LIN {X 0,Y 446.444,Z 326.37,A -85,B 0,C 180,E1 -8665.154,E2 -8665.154} C_VEL
LIN {X 0,Y 446.485,Z 326.372,A -85,B 0,C 180,E1 -8668.179,E2 -8668.179} C_VEL
LIN {X 0,Y 446.42,Z 326.377,A -85,B 0,C 180,E1 -8671.775,E2 -8671.775} C_VEL
LIN {X 0,Y 446.43,Z 326.375,A -85,B 0,C 180,E1 -8674.523,E2 -8674.523} C_VEL
LIN {X 0,Y 446.417,Z 326.381,A -85,B 0,C 180,E1 -8678.08,E2 -8678.08} C_VEL
LIN {X 0,Y 446.439,Z 326.441,A -85,B 0,C 180,E1 -8680.92,E2 -8680.92} C_VEL
LIN {X 0,Y 446.853,Z 329.465,A -85,B 0,C 180,E1 -8683.791,E2 -8683.791} C_VEL
LIN {X 0,Y 447.265,Z 332.288,A -85,B 0,C 180,E1 -8686.288,E2 -8686.288} C_VEL
LIN {X 0,Y 447.313,Z 335.268,A -85,B 0,C 180,E1 -8688.709,E2 -8688.709} C_VEL
LIN {X 0,Y 447.118,Z 339.37,A -85,B 0,C 180,E1 -8691.807,E2 -8691.807} C_VEL
LIN {X 0,Y 446.836,Z 343.714,A -85,B 0,C 180,E1 -8694.873,E2 -8694.873} C_VEL
LIN {X 0,Y 446.563,Z 347.879,A -85,B 0,C 180,E1 -8697.65,E2 -8697.65} C_VEL
LIN {X 0,Y 446.282,Z 352.764,A -85,B 0,C 180,E1 -8700.779,E2 -8700.779} C_VEL
LIN {X 0,Y 446.038,Z 357.892,A -85,B 0,C 180,E1 -8703.913,E2 -8703.913} C_VEL
LIN {X 0,Y 445.811,Z 362.775,A -85,B 0,C 180,E1 -8706.789,E2 -8706.789} C_VEL
LIN {X 0,Y 445.645,Z 367.867,A -85,B 0,C 180,E1 -8709.699,E2 -8709.699} C_VEL
LIN {X 0,Y 445.513,Z 372.967,A -85,B 0,C 180,E1 -8712.559,E2 -8712.559} C_VEL
LIN {X 0,Y 445.479,Z 375.417,A -85,B 0,C 180,E1 -8713.876,E2 -8713.876} C_VEL
LIN {X 0,Y 447.43,Z 386.038,A -85,B 0,C 180,E1 -8714.246,E2 -8714.246} C_VEL
LIN {X 0,Y 448.77,Z 395.709,A -85,B 0,C 180,E1 -8714.676,E2 -8714.676} C_VEL
LIN {X 0,Y 449.202,Z 400.753,A -85,B 0,C 180,E1 -8714.924,E2 -8714.924} C_VEL
LIN {X 0,Y 448.604,Z 412.306,A -85,B 0,C 180,E1 -8715.599,E2 -8715.599} C_VEL
LIN {X 0,Y 448.106,Z 421.585,A -85,B 0,C 180,E1 -8716.278,E2 -8716.278} C_VEL
LIN {X 0,Y 447.61,Z 430.807,A -85,B 0,C 180,E1 -8717.099,E2 -8717.099} C_VEL
LIN {X 0,Y 447.187,Z 439.067,A -85,B 0,C 180,E1 -8717.981,E2 -8717.981} C_VEL
LIN {X 0,Y 446.718,Z 446.286,A -85,B 0,C 180,E1 -8718.888,E2 -8718.888} C_VEL
LIN {X 0,Y 446.391,Z 452.49,A -85,B 0,C 180,E1 -8719.798,E2 -8719.798} C_VEL
LIN {X 0,Y 446.032,Z 459.028,A -85,B 0,C 180,E1 -8720.934,E2 -8720.934} C_VEL
LIN {X 0,Y 445.849,Z 463.531,A -85,B 0,C 180,E1 -8721.844,E2 -8721.844} C_VEL
LIN {X 0,Y 445.576,Z 469.176,A -85,B 0,C 180,E1 -8723.252,E2 -8723.252} C_VEL
LIN {X 0,Y 445.485,Z 473.344,A -85,B 0,C 180,E1 -8724.568,E2 -8724.568} C_VEL
LIN {X 0,Y 445.415,Z 475.709,A -85,B 0,C 180,E1 -8725.475,E2 -8725.475} C_VEL
LIN {X 0,Y 445.433,Z 478.893,A -85,B 0,C 180,E1 -8727.287,E2 -8727.287} C_VEL
LIN {X 0,Y 445.356,Z 479.947,A -85,B 0,C 180,E1 -8728.191,E2 -8728.191} C_VEL
LIN {X 0,Y 445.339,Z 480.535,A -85,B 0,C 180,E1 -8729.096,E2 -8729.096} C_VEL
LIN {X 0,Y 445.339,Z 480.535,A -85,B 0,C 180,E1 -8730.904,E2 -8730.904} C_VEL
LIN {X 0,Y 445.356,Z 479.947,A -85,B 0,C 180,E1 -8731.809,E2 -8731.809} C_VEL
LIN {X 0,Y 445.433,Z 478.893,A -85,B 0,C 180,E1 -8732.713,E2 -8732.713} C_VEL
LIN {X 0,Y 445.415,Z 475.709,A -85,B 0,C 180,E1 -8734.525,E2 -8734.525} C_VEL
LIN {X 0,Y 445.488,Z 471.512,A -85,B 0,C 180,E1 -8736.065,E2 -8736.065} C_VEL
LIN {X 0,Y 445.668,Z 467.361,A -85,B 0,C 180,E1 -8737.248,E2 -8737.248} C_VEL
LIN {X 0,Y 445.96,Z 461.341,A -85,B 0,C 180,E1 -8738.61,E2 -8738.61} C_VEL
LIN {X 0,Y 446.221,Z 455.242,A -85,B 0,C 180,E1 -8739.748,E2 -8739.748} C_VEL
LIN {X 0,Y 446.523,Z 449.541,A -85,B 0,C 180,E1 -8740.657,E2 -8740.657} C_VEL
LIN {X 0,Y 447.057,Z 440.986,A -85,B 0,C 180,E1 -8741.792,E2 -8741.792} C_VEL
LIN {X 0,Y 447.521,Z 432.804,A -85,B 0,C 180,E1 -8742.701,E2 -8742.701} C_VEL
LIN {X 0,Y 447.897,Z 424.583,A -85,B 0,C 180,E1 -8743.472,E2 -8743.472} C_VEL
LIN {X 0,Y 448.394,Z 415.569,A -85,B 0,C 180,E1 -8744.176,E2 -8744.176} C_VEL
LIN {X 0,Y 448.9,Z 405.809,A -85,B 0,C 180,E1 -8744.797,E2 -8744.797} C_VEL
LIN {X 0,Y 449.135,Z 398.298,A -85,B 0,C 180,E1 -8745.195,E2 -8745.195} C_VEL
LIN {X 0,Y 447.528,Z 386.88,A -85,B 0,C 180,E1 -8745.722,E2 -8745.722} C_VEL
LIN {X 0,Y 445.555,Z 376.286,A -85,B 0,C 180,E1 -8746.101,E2 -8746.101} C_VEL
LIN {X 0,Y 445.479,Z 375.413,A -85,B 0,C 180,E1 -8746.126,E2 -8746.126} C_VEL
LIN {X 0,Y 445.613,Z 369.547,A -85,B 0,C 180,E1 -8749.342,E2 -8749.342} C_VEL
LIN {X 0,Y 445.748,Z 364.453,A -85,B 0,C 180,E1 -8752.235,E2 -8752.235} C_VEL
LIN {X 0,Y 445.93,Z 359.403,A -85,B 0,C 180,E1 -8755.184,E2 -8755.184} C_VEL
LIN {X 0,Y 446.214,Z 354.41,A -85,B 0,C 180,E1 -8758.197,E2 -8758.197} C_VEL
LIN {X 0,Y 446.473,Z 349.484,A -85,B 0,C 180,E1 -8761.296,E2 -8761.296} C_VEL
LIN {X 0,Y 446.764,Z 344.641,A -85,B 0,C 180,E1 -8764.493,E2 -8764.493} C_VEL
LIN {X 0,Y 447.042,Z 339.888,A -85,B 0,C 180,E1 -8767.815,E2 -8767.815} C_VEL
LIN {X 0,Y 447.292,Z 335.577,A -85,B 0,C 180,E1 -8771.045,E2 -8771.045} C_VEL
LIN {X 0,Y 447.366,Z 333.745,A -85,B 0,C 180,E1 -8772.494,E2 -8772.494} C_VEL
LIN {X 0,Y 447.054,Z 330.766,A -85,B 0,C 180,E1 -8775.026,E2 -8775.026} C_VEL
LIN {X 0,Y 446.512,Z 326.908,A -85,B 0,C 180,E1 -8778.618,E2 -8778.618} C_VEL
LIN {X 0,Y 446.439,Z 326.441,A -85,B 0,C 180,E1 -8779.08,E2 -8779.08} C_VEL
LIN {X 0,Y 446.417,Z 326.38,A -85,B 0,C 180,E1 -8781.92,E2 -8781.92} C_VEL
LIN {X 0,Y 446.43,Z 326.378,A -85,B 0,C 180,E1 -8785.477,E2 -8785.477} C_VEL
LIN {X 0,Y 446.416,Z 326.374,A -85,B 0,C 180,E1 -8788.699,E2 -8788.699} C_VEL
LIN {X 0,Y 446.485,Z 326.372,A -85,B 0,C 180,E1 -8791.821,E2 -8791.821} C_VEL
LIN {X 0,Y 446.444,Z 326.37,A -85,B 0,C 180,E1 -8794.846,E2 -8794.846} C_VEL
LIN {X 0,Y 446.448,Z 326.371,A -85,B 0,C 180,E1 -8798.245,E2 -8798.245} C_VEL
LIN {X 0,Y 446.453,Z 326.376,A -85,B 0,C 180,E1 -8801.649,E2 -8801.649} C_VEL
LIN {X 0,Y 446.509,Z 326.362,A -85,B 0,C 180,E1 -8804.479,E2 -8804.479} C_VEL
LIN {X 0,Y 446.518,Z 326.361,A -85,B 0,C 180,E1 -8808.193,E2 -8808.193} C_VEL
LIN {X 0,Y 446.6,Z 326.352,A -85,B 0,C 180,E1 -8811.857,E2 -8811.857} C_VEL
LIN {X 0,Y 446.642,Z 326.346,A -85,B 0,C 180,E1 -8814.582,E2 -8814.582} C_VEL
LIN {X 0,Y 446.707,Z 326.344,A -85,B 0,C 180,E1 -8817.294,E2 -8817.294} C_VEL
LIN {X 0,Y 446.792,Z 326.327,A -85,B 0,C 180,E1 -8820,E2 -8820} C_VEL
LIN {X 0,Y 446.708,Z 326.34,A -85,B 0,C 180,E1 -8822.705,E2 -8822.705} C_VEL
LIN {X 0,Y 446.638,Z 326.346,A -85,B 0,C 180,E1 -8826.323,E2 -8826.323} C_VEL
LIN {X 0,Y 446.536,Z 326.365,A -85,B 0,C 180,E1 -8829.055,E2 -8829.055} C_VEL
LIN {X 0,Y 446.52,Z 326.366,A -85,B 0,C 180,E1 -8832.729,E2 -8832.729} C_VEL
LIN {X 0,Y 446.494,Z 326.365,A -85,B 0,C 180,E1 -8836.227,E2 -8836.227} C_VEL
LIN {X 0,Y 446.467,Z 326.368,A -85,B 0,C 180,E1 -8839.303,E2 -8839.303} C_VEL
LIN {X 0,Y 446.416,Z 326.376,A -85,B 0,C 180,E1 -8842.199,E2 -8842.199} C_VEL
LIN {X 0,Y 446.454,Z 326.37,A -85,B 0,C 180,E1 -8845.152,E2 -8845.152} C_VEL
LIN {X 0,Y 446.482,Z 326.369,A -85,B 0,C 180,E1 -8848.178,E2 -8848.178} C_VEL
LIN {X 0,Y 446.417,Z 326.374,A -85,B 0,C 180,E1 -8851.775,E2 -8851.775} C_VEL
LIN {X 0,Y 446.427,Z 326.377,A -85,B 0,C 180,E1 -8854.522,E2 -8854.522} C_VEL
LIN {X 0,Y 446.432,Z 326.377,A -85,B 0,C 180,E1 -8858.082,E2 -8858.082} C_VEL
LIN {X 0,Y 446.444,Z 326.37,A -85,B 0,C 180,E1 -8860.92,E2 -8860.92} C_VEL
LIN {X 0,Y 446.442,Z 326.374,A -85,B 0,C 180,E1 -8863.84,E2 -8863.84} C_VEL
LIN {X 0,Y 446.395,Z 326.379,A -85,B 0,C 180,E1 -8866.403,E2 -8866.403} C_VEL
LIN {X 0,Y 446.464,Z 326.373,A -85,B 0,C 180,E1 -8869.805,E2 -8869.805} C_VEL
LIN {X 0,Y 446.428,Z 326.377,A -85,B 0,C 180,E1 -8872.123,E2 -8872.123} C_VEL
LIN {X 0,Y 446.427,Z 326.375,A -85,B 0,C 180,E1 -8875.477,E2 -8875.477} C_VEL
LIN {X 0,Y 446.413,Z 326.374,A -85,B 0,C 180,E1 -8878.7,E2 -8878.7} C_VEL
LIN {X 0,Y 446.481,Z 326.371,A -85,B 0,C 180,E1 -8881.821,E2 -8881.821} C_VEL
LIN {X 0,Y 446.454,Z 326.369,A -85,B 0,C 180,E1 -8884.848,E2 -8884.848} C_VEL
LIN {X 0,Y 446.444,Z 326.37,A -85,B 0,C 180,E1 -8888.245,E2 -8888.245} C_VEL
LIN {X 0,Y 446.454,Z 326.375,A -85,B 0,C 180,E1 -8891.649,E2 -8891.649} C_VEL
LIN {X 0,Y 446.505,Z 326.366,A -85,B 0,C 180,E1 -8894.48,E2 -8894.48} C_VEL
LIN {X 0,Y 446.514,Z 326.363,A -85,B 0,C 180,E1 -8898.193,E2 -8898.193} C_VEL
LIN {X 0,Y 446.597,Z 326.355,A -85,B 0,C 180,E1 -8901.858,E2 -8901.858} C_VEL
LIN {X 0,Y 446.644,Z 326.349,A -85,B 0,C 180,E1 -8904.583,E2 -8904.583} C_VEL
LIN {X 0,Y 446.616,Z 326.353,A -85,B 0,C 180,E1 -8906.99,E2 -8906.99} C_VEL
LIN {X 0,Y 446.098,Z 326.422,A -85,B 0,C 180,E1 -8907.742,E2 -8907.742} C_VEL
LIN {X 0,Y 443.285,Z 326.777,A -85,B 0,C 180,E1 -8908.965,E2 -8908.965} C_VEL
LIN {X 0,Y 440.802,Z 327.085,A -85,B 0,C 180,E1 -8909.952,E2 -8909.952} C_VEL
LIN {X 0,Y 439.714,Z 327.216,A -85,B 0,C 180,E1 -8910.716,E2 -8910.716} C_VEL
LIN {X 0,Y 439.619,Z 327.225,A -85,B 0,C 180,E1 -8910.975,E2 -8910.975} C_VEL
LIN {X 0,Y 439.653,Z 327.222,A -85,B 0,C 180,E1 -8912.749,E2 -8912.749} C_VEL
LIN {X 0,Y 439.616,Z 327.227,A -85,B 0,C 180,E1 -8916.425,E2 -8916.425} C_VEL
LIN {X 0,Y 439.497,Z 327.24,A -85,B 0,C 180,E1 -8919.202,E2 -8919.202} C_VEL
LIN {X 0,Y 439.462,Z 327.246,A -85,B 0,C 180,E1 -8922.938,E2 -8922.938} C_VEL
LIN {X 0,Y 439.444,Z 327.248,A -85,B 0,C 180,E1 -8926.349,E2 -8926.349} C_VEL
LIN {X 0,Y 439.399,Z 327.247,A -85,B 0,C 180,E1 -8929.626,E2 -8929.626} C_VEL
LIN {X 0,Y 439.361,Z 327.258,A -85,B 0,C 180,E1 -8932.576,E2 -8932.576} C_VEL
LIN {X 0,Y 439.401,Z 327.247,A -85,B 0,C 180,E1 -8935.585,E2 -8935.585} C_VEL
LIN {X 0,Y 439.414,Z 327.249,A -85,B 0,C 180,E1 -8938.674,E2 -8938.674} C_VEL
LIN {X 0,Y 439.367,Z 327.256,A -85,B 0,C 180,E1 -8942.031,E2 -8942.031} C_VEL
LIN {X 0,Y 439.392,Z 327.248,A -85,B 0,C 180,E1 -8945.341,E2 -8945.341} C_VEL
LIN {X 0,Y 439.392,Z 327.25,A -85,B 0,C 180,E1 -8948.594,E2 -8948.594} C_VEL
LIN {X 0,Y 439.395,Z 327.248,A -85,B 0,C 180,E1 -8951.259,E2 -8951.259} C_VEL
LIN {X 0,Y 439.401,Z 327.247,A -85,B 0,C 180,E1 -8954.729,E2 -8954.729} C_VEL
LIN {X 0,Y 439.409,Z 327.253,A -85,B 0,C 180,E1 -8957.798,E2 -8957.798} C_VEL
LIN {X 0,Y 439.446,Z 327.244,A -85,B 0,C 180,E1 -8960.23,E2 -8960.23} C_VEL
LIN {X 0,Y 439.372,Z 327.258,A -85,B 0,C 180,E1 -8963.713,E2 -8963.713} C_VEL
LIN {X 0,Y 439.369,Z 327.252,A -85,B 0,C 180,E1 -8967.054,E2 -8967.054} C_VEL
LIN {X 0,Y 439.379,Z 327.25,A -85,B 0,C 180,E1 -8970.275,E2 -8970.275} C_VEL
LIN {X 0,Y 439.426,Z 327.251,A -85,B 0,C 180,E1 -8973.397,E2 -8973.397} C_VEL
LIN {X 0,Y 439.383,Z 327.249,A -85,B 0,C 180,E1 -8976.43,E2 -8976.43} C_VEL
LIN {X 0,Y 439.387,Z 327.255,A -85,B 0,C 180,E1 -8979.398,E2 -8979.398} C_VEL
LIN {X 0,Y 439.429,Z 327.244,A -85,B 0,C 180,E1 -8982.31,E2 -8982.31} C_VEL
LIN {X 0,Y 439.446,Z 327.249,A -85,B 0,C 180,E1 -8985.174,E2 -8985.174} C_VEL
LIN {X 0,Y 439.482,Z 327.237,A -85,B 0,C 180,E1 -8988.002,E2 -8988.002} C_VEL
LIN {X 0,Y 439.547,Z 327.23,A -85,B 0,C 180,E1 -8991.727,E2 -8991.727} C_VEL
LIN {X 0,Y 439.616,Z 327.223,A -85,B 0,C 180,E1 -8994.496,E2 -8994.496} C_VEL
LIN {X 0,Y 439.635,Z 327.219,A -85,B 0,C 180,E1 -8998.168,E2 -8998.168} C_VEL
LIN {X 0,Y 439.761,Z 327.202,A -85,B 0,C 180,E1 -9000.001,E2 -9000.001} C_VEL
LIN {X 0,Y 439.654,Z 327.223,A -85,B 0,C 180,E1 -9002.749,E2 -9002.749} C_VEL
LIN {X 0,Y 439.611,Z 327.225,A -85,B 0,C 180,E1 -9006.426,E2 -9006.426} C_VEL
LIN {X 0,Y 439.5,Z 327.236,A -85,B 0,C 180,E1 -9009.202,E2 -9009.202} C_VEL
LIN {X 0,Y 439.466,Z 327.242,A -85,B 0,C 180,E1 -9012.938,E2 -9012.938} C_VEL
LIN {X 0,Y 439.446,Z 327.248,A -85,B 0,C 180,E1 -9016.349,E2 -9016.349} C_VEL
LIN {X 0,Y 439.402,Z 327.248,A -85,B 0,C 180,E1 -9019.627,E2 -9019.627} C_VEL
LIN {X 0,Y 439.364,Z 327.255,A -85,B 0,C 180,E1 -9022.576,E2 -9022.576} C_VEL
LIN {X 0,Y 439.398,Z 327.249,A -85,B 0,C 180,E1 -9025.586,E2 -9025.586} C_VEL
LIN {X 0,Y 439.418,Z 327.247,A -85,B 0,C 180,E1 -9028.674,E2 -9028.674} C_VEL
LIN {X 0,Y 439.371,Z 327.258,A -85,B 0,C 180,E1 -9032.031,E2 -9032.031} C_VEL
LIN {X 0,Y 439.395,Z 327.249,A -85,B 0,C 180,E1 -9035.341,E2 -9035.341} C_VEL
LIN {X 0,Y 439.384,Z 327.256,A -85,B 0,C 180,E1 -9038.595,E2 -9038.595} C_VEL
LIN {X 0,Y 439.407,Z 327.254,A -85,B 0,C 180,E1 -9039.85,E2 -9039.85} C_VEL
LIN {X 0,Y 439.501,Z 327.976,A -85,B 0,C 180,E1 -9041.274,E2 -9041.274} C_VEL
LIN {X 0,Y 439.994,Z 331.549,A -85,B 0,C 180,E1 -9044.653,E2 -9044.653} C_VEL
LIN {X 0,Y 440.322,Z 334.513,A -85,B 0,C 180,E1 -9047.241,E2 -9047.241} C_VEL
LIN {X 0,Y 440.206,Z 338.007,A -85,B 0,C 180,E1 -9050.026,E2 -9050.026} C_VEL
LIN {X 0,Y 439.988,Z 342.009,A -85,B 0,C 180,E1 -9053.003,E2 -9053.003} C_VEL
LIN {X 0,Y 439.663,Z 346.592,A -85,B 0,C 180,E1 -9056.225,E2 -9056.225} C_VEL
LIN {X 0,Y 439.366,Z 351.083,A -85,B 0,C 180,E1 -9059.212,E2 -9059.212} C_VEL
LIN {X 0,Y 439.085,Z 356.005,A -85,B 0,C 180,E1 -9062.343,E2 -9062.343} C_VEL
LIN {X 0,Y 438.83,Z 360.988,A -85,B 0,C 180,E1 -9065.393,E2 -9065.393} C_VEL
LIN {X 0,Y 438.634,Z 366.05,A -85,B 0,C 180,E1 -9068.376,E2 -9068.376} C_VEL
LIN {X 0,Y 438.492,Z 371.121,A -85,B 0,C 180,E1 -9071.304,E2 -9071.304} C_VEL
LIN {X 0,Y 438.405,Z 375.252,A -85,B 0,C 180,E1 -9073.607,E2 -9073.607} C_VEL
LIN {X 0,Y 440.56,Z 386.753,A -85,B 0,C 180,E1 -9074.025,E2 -9074.025} C_VEL
LIN {X 0,Y 442.111,Z 398.097,A -85,B 0,C 180,E1 -9074.558,E2 -9074.558} C_VEL
LIN {X 0,Y 442.181,Z 402.591,A -85,B 0,C 180,E1 -9074.796,E2 -9074.796} C_VEL
LIN {X 0,Y 441.714,Z 412.109,A -85,B 0,C 180,E1 -9075.37,E2 -9075.37} C_VEL
LIN {X 0,Y 441.183,Z 421.388,A -85,B 0,C 180,E1 -9076.058,E2 -9076.058} C_VEL
LIN {X 0,Y 440.702,Z 429.36,A -85,B 0,C 180,E1 -9076.764,E2 -9076.764} C_VEL
LIN {X 0,Y 440.364,Z 436.951,A -85,B 0,C 180,E1 -9077.558,E2 -9077.558} C_VEL
LIN {X 0,Y 439.732,Z 446.09,A -85,B 0,C 180,E1 -9078.709,E2 -9078.709} C_VEL
LIN {X 0,Y 439.369,Z 452.294,A -85,B 0,C 180,E1 -9079.633,E2 -9079.633} C_VEL
LIN {X 0,Y 438.994,Z 458.832,A -85,B 0,C 180,E1 -9080.788,E2 -9080.788} C_VEL
LIN {X 0,Y 438.783,Z 463.334,A -85,B 0,C 180,E1 -9081.712,E2 -9081.712} C_VEL
LIN {X 0,Y 438.515,Z 468.824,A -85,B 0,C 180,E1 -9083.096,E2 -9083.096} C_VEL
LIN {X 0,Y 438.385,Z 473.148,A -85,B 0,C 180,E1 -9084.48,E2 -9084.48} C_VEL
LIN {X 0,Y 438.344,Z 475.513,A -85,B 0,C 180,E1 -9085.402,E2 -9085.402} C_VEL
LIN {X 0,Y 438.341,Z 478.697,A -85,B 0,C 180,E1 -9087.243,E2 -9087.243} C_VEL
LIN {X 0,Y 438.279,Z 479.752,A -85,B 0,C 180,E1 -9088.162,E2 -9088.162} C_VEL
LIN {X 0,Y 438.252,Z 480.339,A -85,B 0,C 180,E1 -9089.081,E2 -9089.081} C_VEL
LIN {X 0,Y 438.252,Z 480.339,A -85,B 0,C 180,E1 -9090.919,E2 -9090.919} C_VEL
LIN {X 0,Y 438.279,Z 479.752,A -85,B 0,C 180,E1 -9091.838,E2 -9091.838} C_VEL
LIN {X 0,Y 438.341,Z 478.697,A -85,B 0,C 180,E1 -9092.757,E2 -9092.757} C_VEL
LIN {X 0,Y 438.345,Z 475.513,A -85,B 0,C 180,E1 -9094.598,E2 -9094.598} C_VEL
LIN {X 0,Y 438.445,Z 470.623,A -85,B 0,C 180,E1 -9096.37,E2 -9096.37} C_VEL
LIN {X 0,Y 438.681,Z 465.25,A -85,B 0,C 180,E1 -9097.827,E2 -9097.827} C_VEL
LIN {X 0,Y 438.944,Z 459.988,A -85,B 0,C 180,E1 -9098.981,E2 -9098.981} C_VEL
LIN {X 0,Y 439.282,Z 453.67,A -85,B 0,C 180,E1 -9100.136,E2 -9100.136} C_VEL
LIN {X 0,Y 439.609,Z 447.717,A -85,B 0,C 180,E1 -9101.06,E2 -9101.06} C_VEL
LIN {X 0,Y 440.086,Z 440.79,A -85,B 0,C 180,E1 -9101.982,E2 -9101.982} C_VEL
LIN {X 0,Y 440.579,Z 432.608,A -85,B 0,C 180,E1 -9102.904,E2 -9102.904} C_VEL
LIN {X 0,Y 441.031,Z 423.775,A -85,B 0,C 180,E1 -9103.739,E2 -9103.739} C_VEL
LIN {X 0,Y 441.518,Z 415.374,A -85,B 0,C 180,E1 -9104.401,E2 -9104.401} C_VEL
LIN {X 0,Y 442.038,Z 405.613,A -85,B 0,C 180,E1 -9105.032,E2 -9105.032} C_VEL
LIN {X 0,Y 442.279,Z 399.389,A -85,B 0,C 180,E1 -9105.377,E2 -9105.377} C_VEL
LIN {X 0,Y 440.596,Z 387.272,A -85,B 0,C 180,E1 -9105.956,E2 -9105.956} C_VEL
LIN {X 0,Y 438.525,Z 376.326,A -85,B 0,C 180,E1 -9106.36,E2 -9106.36} C_VEL
LIN {X 0,Y 438.404,Z 375.251,A -85,B 0,C 180,E1 -9106.394,E2 -9106.394} C_VEL
LIN {X 0,Y 438.539,Z 369.408,A -85,B 0,C 180,E1 -9109.666,E2 -9109.666} C_VEL
LIN {X 0,Y 438.694,Z 364.34,A -85,B 0,C 180,E1 -9112.612,E2 -9112.612} C_VEL
LIN {X 0,Y 438.903,Z 359.316,A -85,B 0,C 180,E1 -9115.616,E2 -9115.616} C_VEL
LIN {X 0,Y 439.164,Z 354.348,A -85,B 0,C 180,E1 -9118.691,E2 -9118.691} C_VEL
LIN {X 0,Y 439.483,Z 349.147,A -85,B 0,C 180,E1 -9122.053,E2 -9122.053} C_VEL
LIN {X 0,Y 439.782,Z 344.628,A -85,B 0,C 180,E1 -9125.121,E2 -9125.121} C_VEL
LIN {X 0,Y 440.086,Z 339.911,A -85,B 0,C 180,E1 -9128.522,E2 -9128.522} C_VEL
LIN {X 0,Y 440.336,Z 335.307,A -85,B 0,C 180,E1 -9132.093,E2 -9132.093} C_VEL
LIN {X 0,Y 440.083,Z 332.301,A -85,B 0,C 180,E1 -9134.641,E2 -9134.641} C_VEL
LIN {X 0,Y 439.638,Z 328.89,A -85,B 0,C 180,E1 -9137.824,E2 -9137.824} C_VEL
LIN {X 0,Y 439.462,Z 327.67,A -85,B 0,C 180,E1 -9139.028,E2 -9139.028} C_VEL
LIN {X 0,Y 439.431,Z 327.25,A -85,B 0,C 180,E1 -9140.227,E2 -9140.227} C_VEL
LIN {X 0,Y 439.374,Z 327.257,A -85,B 0,C 180,E1 -9143.712,E2 -9143.712} C_VEL
LIN {X 0,Y 439.373,Z 327.251,A -85,B 0,C 180,E1 -9147.054,E2 -9147.054} C_VEL
LIN {X 0,Y 439.383,Z 327.252,A -85,B 0,C 180,E1 -9150.274,E2 -9150.274} C_VEL
LIN {X 0,Y 439.428,Z 327.246,A -85,B 0,C 180,E1 -9153.396,E2 -9153.396} C_VEL
LIN {X 0,Y 439.384,Z 327.25,A -85,B 0,C 180,E1 -9156.429,E2 -9156.429} C_VEL
LIN {X 0,Y 439.388,Z 327.253,A -85,B 0,C 180,E1 -9159.397,E2 -9159.397} C_VEL
LIN {X 0,Y 439.406,Z 327.247,A -85,B 0,C 180,E1 -9162.308,E2 -9162.308} C_VEL
LIN {X 0,Y 439.449,Z 327.244,A -85,B 0,C 180,E1 -9165.174,E2 -9165.174} C_VEL
LIN {X 0,Y 439.484,Z 327.238,A -85,B 0,C 180,E1 -9168.001,E2 -9168.001} C_VEL
LIN {X 0,Y 439.548,Z 327.232,A -85,B 0,C 180,E1 -9171.726,E2 -9171.726} C_VEL
LIN {X 0,Y 439.617,Z 327.22,A -85,B 0,C 180,E1 -9174.495,E2 -9174.495} C_VEL
LIN {X 0,Y 439.634,Z 327.218,A -85,B 0,C 180,E1 -9178.167,E2 -9178.167} C_VEL
LIN {X 0,Y 439.761,Z 327.202,A -85,B 0,C 180,E1 -9179.999,E2 -9179.999} C_VEL
LIN {X 0,Y 439.655,Z 327.219,A -85,B 0,C 180,E1 -9182.748,E2 -9182.748} C_VEL
LIN {X 0,Y 439.598,Z 327.223,A -85,B 0,C 180,E1 -9186.566,E2 -9186.566} C_VEL
LIN {X 0,Y 439.498,Z 327.239,A -85,B 0,C 180,E1 -9189.201,E2 -9189.201} C_VEL
LIN {X 0,Y 439.464,Z 327.246,A -85,B 0,C 180,E1 -9192.937,E2 -9192.937} C_VEL
LIN {X 0,Y 439.445,Z 327.244,A -85,B 0,C 180,E1 -9196.348,E2 -9196.348} C_VEL
LIN {X 0,Y 439.4,Z 327.247,A -85,B 0,C 180,E1 -9199.626,E2 -9199.626} C_VEL
LIN {X 0,Y 439.362,Z 327.259,A -85,B 0,C 180,E1 -9202.575,E2 -9202.575} C_VEL
LIN {X 0,Y 439.402,Z 327.247,A -85,B 0,C 180,E1 -9205.584,E2 -9205.584} C_VEL
LIN {X 0,Y 439.414,Z 327.251,A -85,B 0,C 180,E1 -9208.673,E2 -9208.673} C_VEL
LIN {X 0,Y 439.368,Z 327.254,A -85,B 0,C 180,E1 -9212.03,E2 -9212.03} C_VEL
LIN {X 0,Y 439.393,Z 327.248,A -85,B 0,C 180,E1 -9215.34,E2 -9215.34} C_VEL
LIN {X 0,Y 439.392,Z 327.251,A -85,B 0,C 180,E1 -9218.593,E2 -9218.593} C_VEL
LIN {X 0,Y 439.401,Z 327.247,A -85,B 0,C 180,E1 -9221.259,E2 -9221.259} C_VEL
LIN {X 0,Y 439.405,Z 327.248,A -85,B 0,C 180,E1 -9224.728,E2 -9224.728} C_VEL
LIN {X 0,Y 439.394,Z 327.253,A -85,B 0,C 180,E1 -9227.796,E2 -9227.796} C_VEL
LIN {X 0,Y 439.445,Z 327.246,A -85,B 0,C 180,E1 -9230.23,E2 -9230.23} C_VEL
LIN {X 0,Y 439.373,Z 327.256,A -85,B 0,C 180,E1 -9233.713,E2 -9233.713} C_VEL
LIN {X 0,Y 439.368,Z 327.252,A -85,B 0,C 180,E1 -9237.054,E2 -9237.054} C_VEL
LIN {X 0,Y 439.379,Z 327.251,A -85,B 0,C 180,E1 -9240.274,E2 -9240.274} C_VEL
LIN {X 0,Y 439.426,Z 327.248,A -85,B 0,C 180,E1 -9243.396,E2 -9243.396} C_VEL
LIN {X 0,Y 439.382,Z 327.249,A -85,B 0,C 180,E1 -9246.429,E2 -9246.429} C_VEL
LIN {X 0,Y 439.386,Z 327.255,A -85,B 0,C 180,E1 -9249.397,E2 -9249.397} C_VEL
LIN {X 0,Y 439.428,Z 327.247,A -85,B 0,C 180,E1 -9252.309,E2 -9252.309} C_VEL
LIN {X 0,Y 439.446,Z 327.248,A -85,B 0,C 180,E1 -9255.174,E2 -9255.174} C_VEL
LIN {X 0,Y 439.48,Z 327.24,A -85,B 0,C 180,E1 -9258.001,E2 -9258.001} C_VEL
LIN {X 0,Y 439.545,Z 327.234,A -85,B 0,C 180,E1 -9261.726,E2 -9261.726} C_VEL
LIN {X 0,Y 439.619,Z 327.224,A -85,B 0,C 180,E1 -9264.496,E2 -9264.496} C_VEL
LIN {X 0,Y 439.633,Z 327.222,A -85,B 0,C 180,E1 -9268.168,E2 -9268.168} C_VEL
LIN {X 0,Y 439.761,Z 327.207,A -85,B 0,C 180,E1 -9270,E2 -9270} C_VEL
LIN {X 0,Y 439.619,Z 327.225,A -85,B 0,C 180,E1 -9270.975,E2 -9270.975} C_VEL
LIN {X 0,Y 438.902,Z 327.313,A -85,B 0,C 180,E1 -9271.739,E2 -9271.739} C_VEL
LIN {X 0,Y 435.923,Z 327.686,A -85,B 0,C 180,E1 -9272.978,E2 -9272.978} C_VEL
LIN {X 0,Y 433.471,Z 327.992,A -85,B 0,C 180,E1 -9273.978,E2 -9273.978} C_VEL
LIN {X 0,Y 432.497,Z 328.113,A -85,B 0,C 180,E1 -9274.753,E2 -9274.753} C_VEL
LIN {X 0,Y 432.46,Z 328.115,A -85,B 0,C 180,E1 -9275.015,E2 -9275.015} C_VEL
LIN {X 0,Y 432.582,Z 328.101,A -85,B 0,C 180,E1 -9277.679,E2 -9277.679} C_VEL
LIN {X 0,Y 432.39,Z 328.125,A -85,B 0,C 180,E1 -9281.247,E2 -9281.247} C_VEL
LIN {X 0,Y 432.371,Z 328.128,A -85,B 0,C 180,E1 -9284.112,E2 -9284.112} C_VEL
LIN {X 0,Y 432.394,Z 328.126,A -85,B 0,C 180,E1 -9287.012,E2 -9287.012} C_VEL
LIN {X 0,Y 432.335,Z 328.129,A -85,B 0,C 180,E1 -9289.96,E2 -9289.96} C_VEL
LIN {X 0,Y 432.315,Z 328.132,A -85,B 0,C 180,E1 -9292.964,E2 -9292.964} C_VEL
LIN {X 0,Y 432.361,Z 328.128,A -85,B 0,C 180,E1 -9296.033,E2 -9296.033} C_VEL
LIN {X 0,Y 432.339,Z 328.127,A -85,B 0,C 180,E1 -9299.188,E2 -9299.188} C_VEL
LIN {X 0,Y 432.319,Z 328.134,A -85,B 0,C 180,E1 -9302.443,E2 -9302.443} C_VEL
LIN {X 0,Y 432.342,Z 328.128,A -85,B 0,C 180,E1 -9305.632,E2 -9305.632} C_VEL
LIN {X 0,Y 432.354,Z 328.126,A -85,B 0,C 180,E1 -9308.718,E2 -9308.718} C_VEL
LIN {X 0,Y 432.362,Z 328.129,A -85,B 0,C 180,E1 -9311.793,E2 -9311.793} C_VEL
LIN {X 0,Y 432.375,Z 328.127,A -85,B 0,C 180,E1 -9315.659,E2 -9315.659} C_VEL
LIN {X 0,Y 432.37,Z 328.124,A -85,B 0,C 180,E1 -9318.392,E2 -9318.392} C_VEL
LIN {X 0,Y 432.347,Z 328.132,A -85,B 0,C 180,E1 -9321.852,E2 -9321.852} C_VEL
LIN {X 0,Y 432.336,Z 328.131,A -85,B 0,C 180,E1 -9325.323,E2 -9325.323} C_VEL
LIN {X 0,Y 432.319,Z 328.129,A -85,B 0,C 180,E1 -9328.654,E2 -9328.654} C_VEL
LIN {X 0,Y 432.379,Z 328.125,A -85,B 0,C 180,E1 -9331.877,E2 -9331.877} C_VEL
LIN {X 0,Y 432.349,Z 328.128,A -85,B 0,C 180,E1 -9334.999,E2 -9334.999} C_VEL
LIN {X 0,Y 432.355,Z 328.125,A -85,B 0,C 180,E1 -9338.046,E2 -9338.046} C_VEL
LIN {X 0,Y 432.384,Z 328.125,A -85,B 0,C 180,E1 -9341.03,E2 -9341.03} C_VEL
LIN {X 0,Y 432.429,Z 328.116,A -85,B 0,C 180,E1 -9343.962,E2 -9343.962} C_VEL
LIN {X 0,Y 432.457,Z 328.113,A -85,B 0,C 180,E1 -9347.804,E2 -9347.804} C_VEL
LIN {X 0,Y 432.491,Z 328.109,A -85,B 0,C 180,E1 -9351.591,E2 -9351.591} C_VEL
LIN {X 0,Y 432.593,Z 328.097,A -85,B 0,C 180,E1 -9354.407,E2 -9354.407} C_VEL
LIN {X 0,Y 432.605,Z 328.094,A -85,B 0,C 180,E1 -9358.139,E2 -9358.139} C_VEL
LIN {X 0,Y 432.731,Z 328.078,A -85,B 0,C 180,E1 -9360.001,E2 -9360.001} C_VEL
LIN {X 0,Y 432.603,Z 328.101,A -85,B 0,C 180,E1 -9362.794,E2 -9362.794} C_VEL
LIN {X 0,Y 432.564,Z 328.105,A -85,B 0,C 180,E1 -9366.531,E2 -9366.531} C_VEL
LIN {X 0,Y 432.443,Z 328.114,A -85,B 0,C 180,E1 -9369.354,E2 -9369.354} C_VEL
LIN {X 0,Y 432.431,Z 328.119,A -85,B 0,C 180,E1 -9372.804,E2 -9372.804} C_VEL
LIN {X 0,Y 432.412,Z 328.125,A -85,B 0,C 180,E1 -9376.479,E2 -9376.479} C_VEL
LIN {X 0,Y 432.338,Z 328.13,A -85,B 0,C 180,E1 -9379.961,E2 -9379.961} C_VEL
LIN {X 0,Y 432.318,Z 328.13,A -85,B 0,C 180,E1 -9382.965,E2 -9382.965} C_VEL
LIN {X 0,Y 432.361,Z 328.13,A -85,B 0,C 180,E1 -9386.033,E2 -9386.033} C_VEL
LIN {X 0,Y 432.343,Z 328.126,A -85,B 0,C 180,E1 -9389.188,E2 -9389.188} C_VEL
LIN {X 0,Y 432.324,Z 328.131,A -85,B 0,C 180,E1 -9392.443,E2 -9392.443} C_VEL
LIN {X 0,Y 432.345,Z 328.13,A -85,B 0,C 180,E1 -9395.632,E2 -9395.632} C_VEL
LIN {X 0,Y 432.351,Z 328.132,A -85,B 0,C 180,E1 -9399.343,E2 -9399.343} C_VEL
LIN {X 0,Y 432.351,Z 328.132,A -85,B 0,C 180,E1 -9400.182,E2 -9400.182} C_VEL
LIN {X 0,Y 432.739,Z 330.94,A -85,B 0,C 180,E1 -9403.044,E2 -9403.044} C_VEL
LIN {X 0,Y 433.184,Z 333.88,A -85,B 0,C 180,E1 -9405.763,E2 -9405.763} C_VEL
LIN {X 0,Y 433.293,Z 336.882,A -85,B 0,C 180,E1 -9408.317,E2 -9408.317} C_VEL
LIN {X 0,Y 433.082,Z 340.511,A -85,B 0,C 180,E1 -9411.164,E2 -9411.164} C_VEL
LIN {X 0,Y 432.821,Z 344.703,A -85,B 0,C 180,E1 -9414.281,E2 -9414.281} C_VEL
LIN {X 0,Y 432.463,Z 349.581,A -85,B 0,C 180,E1 -9417.679,E2 -9417.679} C_VEL
LIN {X 0,Y 432.154,Z 354.289,A -85,B 0,C 180,E1 -9420.799,E2 -9420.799} C_VEL
LIN {X 0,Y 431.901,Z 359.229,A -85,B 0,C 180,E1 -9423.938,E2 -9423.938} C_VEL
LIN {X 0,Y 431.649,Z 364.228,A -85,B 0,C 180,E1 -9426.998,E2 -9426.998} C_VEL
LIN {X 0,Y 431.461,Z 369.271,A -85,B 0,C 180,E1 -9429.997,E2 -9429.997} C_VEL
LIN {X 0,Y 431.336,Z 375.07,A -85,B 0,C 180,E1 -9433.329,E2 -9433.329} C_VEL
LIN {X 0,Y 433.398,Z 386.39,A -85,B 0,C 180,E1 -9433.748,E2 -9433.748} C_VEL
LIN {X 0,Y 434.885,Z 396.601,A -85,B 0,C 180,E1 -9434.235,E2 -9434.235} C_VEL
LIN {X 0,Y 435.434,Z 401.389,A -85,B 0,C 180,E1 -9434.495,E2 -9434.495} C_VEL
LIN {X 0,Y 434.828,Z 411.913,A -85,B 0,C 180,E1 -9435.133,E2 -9435.133} C_VEL
LIN {X 0,Y 434.286,Z 421.192,A -85,B 0,C 180,E1 -9435.832,E2 -9435.832} C_VEL
LIN {X 0,Y 433.717,Z 429.983,A -85,B 0,C 180,E1 -9436.633,E2 -9436.633} C_VEL
LIN {X 0,Y 433.279,Z 438.674,A -85,B 0,C 180,E1 -9437.589,E2 -9437.589} C_VEL
LIN {X 0,Y 432.758,Z 445.894,A -85,B 0,C 180,E1 -9438.525,E2 -9438.525} C_VEL
LIN {X 0,Y 432.348,Z 452.097,A -85,B 0,C 180,E1 -9439.463,E2 -9439.463} C_VEL
LIN {X 0,Y 431.952,Z 458.635,A -85,B 0,C 180,E1 -9440.636,E2 -9440.636} C_VEL
LIN {X 0,Y 431.721,Z 463.137,A -85,B 0,C 180,E1 -9441.575,E2 -9441.575} C_VEL
LIN {X 0,Y 431.437,Z 468.628,A -85,B 0,C 180,E1 -9442.982,E2 -9442.982} C_VEL
LIN {X 0,Y 431.288,Z 472.951,A -85,B 0,C 180,E1 -9444.389,E2 -9444.389} C_VEL
LIN {X 0,Y 431.274,Z 475.318,A -85,B 0,C 180,E1 -9445.326,E2 -9445.326} C_VEL
LIN {X 0,Y 431.236,Z 478.501,A -85,B 0,C 180,E1 -9447.198,E2 -9447.198} C_VEL
LIN {X 0,Y 431.203,Z 479.557,A -85,B 0,C 180,E1 -9448.132,E2 -9448.132} C_VEL
LIN {X 0,Y 431.169,Z 480.144,A -85,B 0,C 180,E1 -9449.066,E2 -9449.066} C_VEL
LIN {X 0,Y 431.169,Z 480.144,A -85,B 0,C 180,E1 -9450.934,E2 -9450.934} C_VEL
LIN {X 0,Y 431.203,Z 479.557,A -85,B 0,C 180,E1 -9451.868,E2 -9451.868} C_VEL
LIN {X 0,Y 431.188,Z 477.113,A -85,B 0,C 180,E1 -9453.738,E2 -9453.738} C_VEL
LIN {X 0,Y 431.299,Z 474.168,A -85,B 0,C 180,E1 -9455.142,E2 -9455.142} C_VEL
LIN {X 0,Y 431.378,Z 470.181,A -85,B 0,C 180,E1 -9456.548,E2 -9456.548} C_VEL
LIN {X 0,Y 431.608,Z 465.053,A -85,B 0,C 180,E1 -9457.956,E2 -9457.956} C_VEL
LIN {X 0,Y 431.881,Z 459.79,A -85,B 0,C 180,E1 -9459.129,E2 -9459.129} C_VEL
LIN {X 0,Y 432.248,Z 453.473,A -85,B 0,C 180,E1 -9460.303,E2 -9460.303} C_VEL
LIN {X 0,Y 432.626,Z 447.52,A -85,B 0,C 180,E1 -9461.241,E2 -9461.241} C_VEL
LIN {X 0,Y 433.13,Z 440.594,A -85,B 0,C 180,E1 -9462.177,E2 -9462.177} C_VEL
LIN {X 0,Y 433.624,Z 432.411,A -85,B 0,C 180,E1 -9463.115,E2 -9463.115} C_VEL
LIN {X 0,Y 434.062,Z 424.486,A -85,B 0,C 180,E1 -9463.884,E2 -9463.884} C_VEL
LIN {X 0,Y 434.627,Z 415.177,A -85,B 0,C 180,E1 -9464.635,E2 -9464.635} C_VEL
LIN {X 0,Y 435.158,Z 405.416,A -85,B 0,C 180,E1 -9465.275,E2 -9465.275} C_VEL
LIN {X 0,Y 435.403,Z 400.359,A -85,B 0,C 180,E1 -9465.566,E2 -9465.566} C_VEL
LIN {X 0,Y 433.548,Z 387.275,A -85,B 0,C 180,E1 -9466.215,E2 -9466.215} C_VEL
LIN {X 0,Y 431.601,Z 376.875,A -85,B 0,C 180,E1 -9466.613,E2 -9466.613} C_VEL
LIN {X 0,Y 431.334,Z 375.07,A -85,B 0,C 180,E1 -9466.671,E2 -9466.671} C_VEL
LIN {X 0,Y 431.462,Z 369.269,A -85,B 0,C 180,E1 -9470.003,E2 -9470.003} C_VEL
LIN {X 0,Y 431.649,Z 364.227,A -85,B 0,C 180,E1 -9473.002,E2 -9473.002} C_VEL
LIN {X 0,Y 431.901,Z 359.227,A -85,B 0,C 180,E1 -9476.062,E2 -9476.062} C_VEL
LIN {X 0,Y 432.155,Z 354.285,A -85,B 0,C 180,E1 -9479.201,E2 -9479.201} C_VEL
LIN {X 0,Y 432.472,Z 349.414,A -85,B 0,C 180,E1 -9482.43,E2 -9482.43} C_VEL
LIN {X 0,Y 432.782,Z 344.619,A -85,B 0,C 180,E1 -9485.775,E2 -9485.775} C_VEL
LIN {X 0,Y 433.07,Z 340.486,A -85,B 0,C 180,E1 -9488.834,E2 -9488.834} C_VEL
LIN {X 0,Y 433.295,Z 336.789,A -85,B 0,C 180,E1 -9491.744,E2 -9491.744} C_VEL
LIN {X 0,Y 433.098,Z 333.639,A -85,B 0,C 180,E1 -9494.438,E2 -9494.438} C_VEL
LIN {X 0,Y 432.738,Z 330.9,A -85,B 0,C 180,E1 -9496.991,E2 -9496.991} C_VEL
LIN {X 0,Y 432.351,Z 328.132,A -85,B 0,C 180,E1 -9499.818,E2 -9499.818} C_VEL
LIN {X 0,Y 432.307,Z 328.136,A -85,B 0,C 180,E1 -9503.022,E2 -9503.022} C_VEL
LIN {X 0,Y 432.36,Z 328.132,A -85,B 0,C 180,E1 -9505.996,E2 -9505.996} C_VEL
LIN {X 0,Y 432.348,Z 328.128,A -85,B 0,C 180,E1 -9509.489,E2 -9509.489} C_VEL
LIN {X 0,Y 432.391,Z 328.12,A -85,B 0,C 180,E1 -9512.928,E2 -9512.928} C_VEL
LIN {X 0,Y 432.368,Z 328.127,A -85,B 0,C 180,E1 -9516.023,E2 -9516.023} C_VEL
LIN {X 0,Y 432.35,Z 328.126,A -85,B 0,C 180,E1 -9519.046,E2 -9519.046} C_VEL
LIN {X 0,Y 432.361,Z 328.127,A -85,B 0,C 180,E1 -9522.01,E2 -9522.01} C_VEL
LIN {X 0,Y 432.396,Z 328.121,A -85,B 0,C 180,E1 -9524.926,E2 -9524.926} C_VEL
LIN {X 0,Y 432.459,Z 328.115,A -85,B 0,C 180,E1 -9527.803,E2 -9527.803} C_VEL
LIN {X 0,Y 432.492,Z 328.113,A -85,B 0,C 180,E1 -9531.59,E2 -9531.59} C_VEL
LIN {X 0,Y 432.594,Z 328.095,A -85,B 0,C 180,E1 -9534.406,E2 -9534.406} C_VEL
LIN {X 0,Y 432.604,Z 328.094,A -85,B 0,C 180,E1 -9538.138,E2 -9538.138} C_VEL
LIN {X 0,Y 432.731,Z 328.078,A -85,B 0,C 180,E1 -9539.999,E2 -9539.999} C_VEL
LIN {X 0,Y 432.604,Z 328.097,A -85,B 0,C 180,E1 -9542.793,E2 -9542.793} C_VEL
LIN {X 0,Y 432.562,Z 328.101,A -85,B 0,C 180,E1 -9546.557,E2 -9546.557} C_VEL
LIN {X 0,Y 432.441,Z 328.117,A -85,B 0,C 180,E1 -9549.353,E2 -9549.353} C_VEL
LIN {X 0,Y 432.429,Z 328.122,A -85,B 0,C 180,E1 -9552.803,E2 -9552.803} C_VEL
LIN {X 0,Y 432.411,Z 328.122,A -85,B 0,C 180,E1 -9556.478,E2 -9556.478} C_VEL
LIN {X 0,Y 432.337,Z 328.128,A -85,B 0,C 180,E1 -9559.96,E2 -9559.96} C_VEL
LIN {X 0,Y 432.316,Z 328.133,A -85,B 0,C 180,E1 -9562.964,E2 -9562.964} C_VEL
LIN {X 0,Y 432.361,Z 328.126,A -85,B 0,C 180,E1 -9566.032,E2 -9566.032} C_VEL
LIN {X 0,Y 432.34,Z 328.127,A -85,B 0,C 180,E1 -9569.187,E2 -9569.187} C_VEL
LIN {X 0,Y 432.32,Z 328.136,A -85,B 0,C 180,E1 -9572.443,E2 -9572.443} C_VEL
LIN {X 0,Y 432.342,Z 328.127,A -85,B 0,C 180,E1 -9575.632,E2 -9575.632} C_VEL
LIN {X 0,Y 432.354,Z 328.127,A -85,B 0,C 180,E1 -9578.717,E2 -9578.717} C_VEL
LIN {X 0,Y 432.37,Z 328.126,A -85,B 0,C 180,E1 -9581.792,E2 -9581.792} C_VEL
LIN {X 0,Y 432.375,Z 328.127,A -85,B 0,C 180,E1 -9584.341,E2 -9584.341} C_VEL
LIN {X 0,Y 432.362,Z 328.129,A -85,B 0,C 180,E1 -9588.207,E2 -9588.207} C_VEL
LIN {X 0,Y 432.354,Z 328.126,A -85,B 0,C 180,E1 -9591.282,E2 -9591.282} C_VEL
LIN {X 0,Y 432.342,Z 328.128,A -85,B 0,C 180,E1 -9594.368,E2 -9594.368} C_VEL
LIN {X 0,Y 432.319,Z 328.134,A -85,B 0,C 180,E1 -9597.557,E2 -9597.557} C_VEL
LIN {X 0,Y 432.339,Z 328.127,A -85,B 0,C 180,E1 -9600.812,E2 -9600.812} C_VEL
LIN {X 0,Y 432.361,Z 328.128,A -85,B 0,C 180,E1 -9603.967,E2 -9603.967} C_VEL
LIN {X 0,Y 432.315,Z 328.132,A -85,B 0,C 180,E1 -9607.036,E2 -9607.036} C_VEL
LIN {X 0,Y 432.383,Z 328.122,A -85,B 0,C 180,E1 -9610.515,E2 -9610.515} C_VEL
LIN {X 0,Y 432.427,Z 328.121,A -85,B 0,C 180,E1 -9613.961,E2 -9613.961} C_VEL
LIN {X 0,Y 432.456,Z 328.116,A -85,B 0,C 180,E1 -9617.803,E2 -9617.803} C_VEL
LIN {X 0,Y 432.489,Z 328.113,A -85,B 0,C 180,E1 -9621.59,E2 -9621.59} C_VEL
LIN {X 0,Y 432.596,Z 328.099,A -85,B 0,C 180,E1 -9624.406,E2 -9624.406} C_VEL
LIN {X 0,Y 432.603,Z 328.097,A -85,B 0,C 180,E1 -9628.138,E2 -9628.138} C_VEL
LIN {X 0,Y 432.73,Z 328.083,A -85,B 0,C 180,E1 -9630,E2 -9630} C_VEL
LIN {X 0,Y 432.602,Z 328.1,A -85,B 0,C 180,E1 -9632.794,E2 -9632.794} C_VEL
LIN {X 0,Y 432.46,Z 328.115,A -85,B 0,C 180,E1 -9635.015,E2 -9635.015} C_VEL
LIN {X 0,Y 431.9,Z 328.186,A -85,B 0,C 180,E1 -9635.793,E2 -9635.793} C_VEL
LIN {X 0,Y 429.055,Z 328.542,A -85,B 0,C 180,E1 -9637.058,E2 -9637.058} C_VEL
LIN {X 0,Y 426.572,Z 328.85,A -85,B 0,C 180,E1 -9638.079,E2 -9638.079} C_VEL
LIN {X 0,Y 425.491,Z 328.986,A -85,B 0,C 180,E1 -9638.869,E2 -9638.869} C_VEL
LIN {X 0,Y 425.4,Z 328.995,A -85,B 0,C 180,E1 -9639.137,E2 -9639.137} C_VEL
LIN {X 0,Y 425.39,Z 328.999,A -85,B 0,C 180,E1 -9642.904,E2 -9642.904} C_VEL
LIN {X 0,Y 425.358,Z 329.004,A -85,B 0,C 180,E1 -9646.605,E2 -9646.605} C_VEL
LIN {X 0,Y 425.325,Z 329.001,A -85,B 0,C 180,E1 -9649.636,E2 -9649.636} C_VEL
LIN {X 0,Y 425.303,Z 329.003,A -85,B 0,C 180,E1 -9653.365,E2 -9653.365} C_VEL
LIN {X 0,Y 425.345,Z 329,A -85,B 0,C 180,E1 -9656.845,E2 -9656.845} C_VEL
LIN {X 0,Y 425.287,Z 329.007,A -85,B 0,C 180,E1 -9659.72,E2 -9659.72} C_VEL
LIN {X 0,Y 425.278,Z 329.007,A -85,B 0,C 180,E1 -9663.048,E2 -9663.048} C_VEL
LIN {X 0,Y 425.281,Z 329.011,A -85,B 0,C 180,E1 -9665.929,E2 -9665.929} C_VEL
LIN {X 0,Y 425.307,Z 329.003,A -85,B 0,C 180,E1 -9669.046,E2 -9669.046} C_VEL
LIN {X 0,Y 425.311,Z 329.01,A -85,B 0,C 180,E1 -9671.962,E2 -9671.962} C_VEL
LIN {X 0,Y 425.31,Z 329.003,A -85,B 0,C 180,E1 -9675.279,E2 -9675.279} C_VEL
LIN {X 0,Y 425.306,Z 329.003,A -85,B 0,C 180,E1 -9678.626,E2 -9678.626} C_VEL
LIN {X 0,Y 425.318,Z 329.002,A -85,B 0,C 180,E1 -9681.104,E2 -9681.104} C_VEL
LIN {X 0,Y 425.296,Z 329.004,A -85,B 0,C 180,E1 -9684.665,E2 -9684.665} C_VEL
LIN {X 0,Y 425.262,Z 329.01,A -85,B 0,C 180,E1 -9688.074,E2 -9688.074} C_VEL
LIN {X 0,Y 425.328,Z 329.006,A -85,B 0,C 180,E1 -9691.368,E2 -9691.368} C_VEL
LIN {X 0,Y 425.292,Z 329.005,A -85,B 0,C 180,E1 -9694.555,E2 -9694.555} C_VEL
LIN {X 0,Y 425.285,Z 329.009,A -85,B 0,C 180,E1 -9697.662,E2 -9697.662} C_VEL
LIN {X 0,Y 425.36,Z 328.997,A -85,B 0,C 180,E1 -9700.705,E2 -9700.705} C_VEL
LIN {X 0,Y 425.386,Z 328.995,A -85,B 0,C 180,E1 -9703.689,E2 -9703.689} C_VEL
LIN {X 0,Y 425.41,Z 328.992,A -85,B 0,C 180,E1 -9707.599,E2 -9707.599} C_VEL
LIN {X 0,Y 425.441,Z 328.989,A -85,B 0,C 180,E1 -9711.45,E2 -9711.45} C_VEL
LIN {X 0,Y 425.549,Z 328.974,A -85,B 0,C 180,E1 -9714.314,E2 -9714.314} C_VEL
LIN {X 0,Y 425.575,Z 328.97,A -85,B 0,C 180,E1 -9718.108,E2 -9718.108} C_VEL
LIN {X 0,Y 425.701,Z 328.954,A -85,B 0,C 180,E1 -9720.001,E2 -9720.001} C_VEL
LIN {X 0,Y 425.555,Z 328.978,A -85,B 0,C 180,E1 -9722.84,E2 -9722.84} C_VEL
LIN {X 0,Y 425.523,Z 328.983,A -85,B 0,C 180,E1 -9726.639,E2 -9726.639} C_VEL
LIN {X 0,Y 425.401,Z 328.991,A -85,B 0,C 180,E1 -9729.51,E2 -9729.51} C_VEL
LIN {X 0,Y 425.393,Z 328.995,A -85,B 0,C 180,E1 -9732.904,E2 -9732.904} C_VEL
LIN {X 0,Y 425.361,Z 329.001,A -85,B 0,C 180,E1 -9736.605,E2 -9736.605} C_VEL
LIN {X 0,Y 425.328,Z 329.001,A -85,B 0,C 180,E1 -9739.636,E2 -9739.636} C_VEL
LIN {X 0,Y 425.288,Z 329.012,A -85,B 0,C 180,E1 -9742.339,E2 -9742.339} C_VEL
LIN {X 0,Y 425.291,Z 329.005,A -85,B 0,C 180,E1 -9745.446,E2 -9745.446} C_VEL
LIN {X 0,Y 425.349,Z 328.999,A -85,B 0,C 180,E1 -9747.558,E2 -9747.558} C_VEL
LIN {X 0,Y 425.288,Z 329.006,A -85,B 0,C 180,E1 -9750.817,E2 -9750.817} C_VEL
LIN {X 0,Y 425.312,Z 329.01,A -85,B 0,C 180,E1 -9754.288,E2 -9754.288} C_VEL
LIN {X 0,Y 425.281,Z 329.013,A -85,B 0,C 180,E1 -9757.695,E2 -9757.695} C_VEL
LIN {X 0,Y 425.338,Z 329.201,A -85,B 0,C 180,E1 -9760.122,E2 -9760.122} C_VEL
LIN {X 0,Y 425.774,Z 332.474,A -85,B 0,C 180,E1 -9763.425,E2 -9763.425} C_VEL
LIN {X 0,Y 426.208,Z 335.827,A -85,B 0,C 180,E1 -9766.515,E2 -9766.515} C_VEL
LIN {X 0,Y 426.178,Z 339.171,A -85,B 0,C 180,E1 -9769.339,E2 -9769.339} C_VEL
LIN {X 0,Y 425.967,Z 343.056,A -85,B 0,C 180,E1 -9772.377,E2 -9772.377} C_VEL
LIN {X 0,Y 425.613,Z 347.538,A -85,B 0,C 180,E1 -9775.653,E2 -9775.653} C_VEL
LIN {X 0,Y 425.354,Z 350.985,A -85,B 0,C 180,E1 -9778.081,E2 -9778.081} C_VEL
LIN {X 0,Y 425.035,Z 355.86,A -85,B 0,C 180,E1 -9781.346,E2 -9781.346} C_VEL
LIN {X 0,Y 424.742,Z 360.802,A -85,B 0,C 180,E1 -9784.519,E2 -9784.519} C_VEL
LIN {X 0,Y 424.524,Z 365.783,A -85,B 0,C 180,E1 -9787.619,E2 -9787.619} C_VEL
LIN {X 0,Y 424.341,Z 370.972,A -85,B 0,C 180,E1 -9790.743,E2 -9790.743} C_VEL
LIN {X 0,Y 424.255,Z 374.888,A -85,B 0,C 180,E1 -9793.047,E2 -9793.047} C_VEL
LIN {X 0,Y 426.284,Z 385.803,A -85,B 0,C 180,E1 -9793.456,E2 -9793.456} C_VEL
LIN {X 0,Y 427.732,Z 395.262,A -85,B 0,C 180,E1 -9793.91,E2 -9793.91} C_VEL
LIN {X 0,Y 428.504,Z 402.269,A -85,B 0,C 180,E1 -9794.303,E2 -9794.303} C_VEL
LIN {X 0,Y 427.951,Z 411.717,A -85,B 0,C 180,E1 -9794.888,E2 -9794.888} C_VEL
LIN {X 0,Y 427.377,Z 420.995,A -85,B 0,C 180,E1 -9795.598,E2 -9795.598} C_VEL
LIN {X 0,Y 426.797,Z 429.787,A -85,B 0,C 180,E1 -9796.412,E2 -9796.412} C_VEL
LIN {X 0,Y 426.311,Z 438.478,A -85,B 0,C 180,E1 -9797.383,E2 -9797.383} C_VEL
LIN {X 0,Y 425.785,Z 445.697,A -85,B 0,C 180,E1 -9798.335,E2 -9798.335} C_VEL
LIN {X 0,Y 425.317,Z 451.899,A -85,B 0,C 180,E1 -9799.287,E2 -9799.287} C_VEL
LIN {X 0,Y 424.894,Z 458.437,A -85,B 0,C 180,E1 -9800.479,E2 -9800.479} C_VEL
LIN {X 0,Y 424.683,Z 462.941,A -85,B 0,C 180,E1 -9801.435,E2 -9801.435} C_VEL
LIN {X 0,Y 424.364,Z 468.431,A -85,B 0,C 180,E1 -9802.865,E2 -9802.865} C_VEL
LIN {X 0,Y 424.196,Z 472.754,A -85,B 0,C 180,E1 -9804.295,E2 -9804.295} C_VEL
LIN {X 0,Y 424.203,Z 475.122,A -85,B 0,C 180,E1 -9805.248,E2 -9805.248} C_VEL
LIN {X 0,Y 424.132,Z 478.305,A -85,B 0,C 180,E1 -9807.151,E2 -9807.151} C_VEL
LIN {X 0,Y 424.129,Z 479.362,A -85,B 0,C 180,E1 -9808.101,E2 -9808.101} C_VEL
LIN {X 0,Y 424.089,Z 479.948,A -85,B 0,C 180,E1 -9809.05,E2 -9809.05} C_VEL
LIN {X 0,Y 424.089,Z 479.948,A -85,B 0,C 180,E1 -9810.95,E2 -9810.95} C_VEL
LIN {X 0,Y 424.129,Z 479.362,A -85,B 0,C 180,E1 -9811.899,E2 -9811.899} C_VEL
LIN {X 0,Y 424.1,Z 476.917,A -85,B 0,C 180,E1 -9813.801,E2 -9813.801} C_VEL
LIN {X 0,Y 424.212,Z 473.972,A -85,B 0,C 180,E1 -9815.228,E2 -9815.228} C_VEL
LIN {X 0,Y 424.303,Z 469.985,A -85,B 0,C 180,E1 -9816.658,E2 -9816.658} C_VEL
LIN {X 0,Y 424.552,Z 464.856,A -85,B 0,C 180,E1 -9818.089,E2 -9818.089} C_VEL
LIN {X 0,Y 424.834,Z 459.594,A -85,B 0,C 180,E1 -9819.282,E2 -9819.282} C_VEL
LIN {X 0,Y 425.221,Z 453.276,A -85,B 0,C 180,E1 -9820.475,E2 -9820.475} C_VEL
LIN {X 0,Y 425.655,Z 447.324,A -85,B 0,C 180,E1 -9821.428,E2 -9821.428} C_VEL
LIN {X 0,Y 426.172,Z 440.397,A -85,B 0,C 180,E1 -9822.379,E2 -9822.379} C_VEL
LIN {X 0,Y 426.671,Z 432.214,A -85,B 0,C 180,E1 -9823.333,E2 -9823.333} C_VEL
LIN {X 0,Y 427.202,Z 423.424,A -85,B 0,C 180,E1 -9824.189,E2 -9824.189} C_VEL
LIN {X 0,Y 427.74,Z 414.981,A -85,B 0,C 180,E1 -9824.876,E2 -9824.876} C_VEL
LIN {X 0,Y 428.247,Z 406.262,A -85,B 0,C 180,E1 -9825.465,E2 -9825.465} C_VEL
LIN {X 0,Y 428.399,Z 400.251,A -85,B 0,C 180,E1 -9825.822,E2 -9825.822} C_VEL
LIN {X 0,Y 426.514,Z 387.197,A -85,B 0,C 180,E1 -9826.486,E2 -9826.486} C_VEL
LIN {X 0,Y 424.396,Z 376.106,A -85,B 0,C 180,E1 -9826.917,E2 -9826.917} C_VEL
LIN {X 0,Y 424.253,Z 374.888,A -85,B 0,C 180,E1 -9826.953,E2 -9826.953} C_VEL
LIN {X 0,Y 424.392,Z 369.13,A -85,B 0,C 180,E1 -9830.35,E2 -9830.35} C_VEL
LIN {X 0,Y 424.586,Z 364.11,A -85,B 0,C 180,E1 -9833.407,E2 -9833.407} C_VEL
LIN {X 0,Y 424.893,Z 358.833,A -85,B 0,C 180,E1 -9836.722,E2 -9836.722} C_VEL
LIN {X 0,Y 425.133,Z 354.222,A -85,B 0,C 180,E1 -9839.732,E2 -9839.732} C_VEL
LIN {X 0,Y 425.47,Z 349.371,A -85,B 0,C 180,E1 -9843.031,E2 -9843.031} C_VEL
LIN {X 0,Y 425.761,Z 345.197,A -85,B 0,C 180,E1 -9846.017,E2 -9846.017} C_VEL
LIN {X 0,Y 426.073,Z 341.041,A -85,B 0,C 180,E1 -9849.171,E2 -9849.171} C_VEL
LIN {X 0,Y 426.256,Z 337.405,A -85,B 0,C 180,E1 -9852.102,E2 -9852.102} C_VEL
LIN {X 0,Y 426.035,Z 334.326,A -85,B 0,C 180,E1 -9854.818,E2 -9854.818} C_VEL
LIN {X 0,Y 425.571,Z 331.02,A -85,B 0,C 180,E1 -9857.999,E2 -9857.999} C_VEL
LIN {X 0,Y 425.338,Z 329.202,A -85,B 0,C 180,E1 -9859.878,E2 -9859.878} C_VEL
LIN {X 0,Y 425.279,Z 329.013,A -85,B 0,C 180,E1 -9862.488,E2 -9862.488} C_VEL
LIN {X 0,Y 425.308,Z 329.011,A -85,B 0,C 180,E1 -9865.817,E2 -9865.817} C_VEL
LIN {X 0,Y 425.291,Z 329.005,A -85,B 0,C 180,E1 -9869.238,E2 -9869.238} C_VEL
LIN {X 0,Y 425.349,Z 328.999,A -85,B 0,C 180,E1 -9872.442,E2 -9872.442} C_VEL
LIN {X 0,Y 425.348,Z 329.003,A -85,B 0,C 180,E1 -9875.601,E2 -9875.601} C_VEL
LIN {X 0,Y 425.293,Z 329.005,A -85,B 0,C 180,E1 -9878.681,E2 -9878.681} C_VEL
LIN {X 0,Y 425.322,Z 329.007,A -85,B 0,C 180,E1 -9881.702,E2 -9881.702} C_VEL
LIN {X 0,Y 425.349,Z 328.998,A -85,B 0,C 180,E1 -9884.67,E2 -9884.67} C_VEL
LIN {X 0,Y 425.412,Z 328.996,A -85,B 0,C 180,E1 -9887.598,E2 -9887.598} C_VEL
LIN {X 0,Y 425.442,Z 328.993,A -85,B 0,C 180,E1 -9891.449,E2 -9891.449} C_VEL
LIN {X 0,Y 425.55,Z 328.973,A -85,B 0,C 180,E1 -9894.313,E2 -9894.313} C_VEL
LIN {X 0,Y 425.574,Z 328.97,A -85,B 0,C 180,E1 -9898.107,E2 -9898.107} C_VEL
LIN {X 0,Y 425.701,Z 328.954,A -85,B 0,C 180,E1 -9899.999,E2 -9899.999} C_VEL
LIN {X 0,Y 425.555,Z 328.976,A -85,B 0,C 180,E1 -9902.839,E2 -9902.839} C_VEL
LIN {X 0,Y 425.522,Z 328.979,A -85,B 0,C 180,E1 -9906.638,E2 -9906.638} C_VEL
LIN {X 0,Y 425.399,Z 328.993,A -85,B 0,C 180,E1 -9909.509,E2 -9909.509} C_VEL
LIN {X 0,Y 425.392,Z 328.999,A -85,B 0,C 180,E1 -9912.903,E2 -9912.903} C_VEL
LIN {X 0,Y 425.359,Z 329.001,A -85,B 0,C 180,E1 -9916.605,E2 -9916.605} C_VEL
LIN {X 0,Y 425.326,Z 329,A -85,B 0,C 180,E1 -9919.635,E2 -9919.635} C_VEL
LIN {X 0,Y 425.285,Z 329.009,A -85,B 0,C 180,E1 -9922.338,E2 -9922.338} C_VEL
LIN {X 0,Y 425.292,Z 329.005,A -85,B 0,C 180,E1 -9925.445,E2 -9925.445} C_VEL
LIN {X 0,Y 425.328,Z 329.006,A -85,B 0,C 180,E1 -9928.632,E2 -9928.632} C_VEL
LIN {X 0,Y 425.262,Z 329.01,A -85,B 0,C 180,E1 -9931.926,E2 -9931.926} C_VEL
LIN {X 0,Y 425.297,Z 329.004,A -85,B 0,C 180,E1 -9935.335,E2 -9935.335} C_VEL
LIN {X 0,Y 425.307,Z 329.003,A -85,B 0,C 180,E1 -9939.045,E2 -9939.045} C_VEL
LIN {X 0,Y 425.328,Z 329.002,A -85,B 0,C 180,E1 -9942.646,E2 -9942.646} C_VEL
LIN {X 0,Y 425.293,Z 329.005,A -85,B 0,C 180,E1 -9945.281,E2 -9945.281} C_VEL
LIN {X 0,Y 425.3,Z 329.005,A -85,B 0,C 180,E1 -9948.625,E2 -9948.625} C_VEL
LIN {X 0,Y 425.318,Z 329.002,A -85,B 0,C 180,E1 -9951.104,E2 -9951.104} C_VEL
LIN {X 0,Y 425.297,Z 329.004,A -85,B 0,C 180,E1 -9954.664,E2 -9954.664} C_VEL
LIN {X 0,Y 425.262,Z 329.012,A -85,B 0,C 180,E1 -9958.073,E2 -9958.073} C_VEL
LIN {X 0,Y 425.327,Z 329.004,A -85,B 0,C 180,E1 -9961.368,E2 -9961.368} C_VEL
LIN {X 0,Y 425.292,Z 329.005,A -85,B 0,C 180,E1 -9964.555,E2 -9964.555} C_VEL
LIN {X 0,Y 425.284,Z 329.012,A -85,B 0,C 180,E1 -9967.661,E2 -9967.661} C_VEL
LIN {X 0,Y 425.358,Z 328.999,A -85,B 0,C 180,E1 -9970.704,E2 -9970.704} C_VEL
LIN {X 0,Y 425.385,Z 328.999,A -85,B 0,C 180,E1 -9973.688,E2 -9973.688} C_VEL
LIN {X 0,Y 425.408,Z 328.995,A -85,B 0,C 180,E1 -9977.598,E2 -9977.598} C_VEL
LIN {X 0,Y 425.439,Z 328.992,A -85,B 0,C 180,E1 -9981.45,E2 -9981.45} C_VEL
LIN {X 0,Y 425.552,Z 328.976,A -85,B 0,C 180,E1 -9984.313,E2 -9984.313} C_VEL
LIN {X 0,Y 425.572,Z 328.973,A -85,B 0,C 180,E1 -9988.107,E2 -9988.107} C_VEL
LIN {X 0,Y 425.7,Z 328.959,A -85,B 0,C 180,E1 -9990,E2 -9990} C_VEL
LIN {X 0,Y 425.554,Z 328.978,A -85,B 0,C 180,E1 -9992.84,E2 -9992.84} C_VEL
LIN {X 0,Y 425.528,Z 328.981,A -85,B 0,C 180,E1 -9996.639,E2 -9996.639} C_VEL
LIN {X 0,Y 425.4,Z 328.995,A -85,B 0,C 180,E1 -9999.137,E2 -9999.137} C_VEL
LIN {X 0,Y 424.727,Z 329.081,A -85,B 0,C 180,E1 -9999.927,E2 -9999.927} C_VEL
LIN {X 0,Y 421.88,Z 329.437,A -85,B 0,C 180,E1 -10001.21,E2 -10001.21} C_VEL
LIN {X 0,Y 419.464,Z 329.738,A -85,B 0,C 180,E1 -10002.247,E2 -10002.247} C_VEL
LIN {X 0,Y 418.413,Z 329.868,A -85,B 0,C 180,E1 -10003.047,E2 -10003.047} C_VEL
LIN {X 0,Y 418.32,Z 329.878,A -85,B 0,C 180,E1 -10003.319,E2 -10003.319} C_VEL
LIN {X 0,Y 418.309,Z 329.881,A -85,B 0,C 180,E1 -10006.736,E2 -10006.736} C_VEL
LIN {X 0,Y 418.267,Z 329.881,A -85,B 0,C 180,E1 -10009.79,E2 -10009.79} C_VEL
LIN {X 0,Y 418.234,Z 329.888,A -85,B 0,C 180,E1 -10012.736,E2 -10012.736} C_VEL
LIN {X 0,Y 418.267,Z 329.882,A -85,B 0,C 180,E1 -10015.904,E2 -10015.904} C_VEL
LIN {X 0,Y 418.261,Z 329.881,A -85,B 0,C 180,E1 -10019.162,E2 -10019.162} C_VEL
LIN {X 0,Y 418.254,Z 329.882,A -85,B 0,C 180,E1 -10022.844,E2 -10022.844} C_VEL
LIN {X 0,Y 418.245,Z 329.888,A -85,B 0,C 180,E1 -10026.239,E2 -10026.239} C_VEL
LIN {X 0,Y 418.261,Z 329.884,A -85,B 0,C 180,E1 -10029.681,E2 -10029.681} C_VEL
LIN {X 0,Y 418.241,Z 329.886,A -85,B 0,C 180,E1 -10032.324,E2 -10032.324} C_VEL
LIN {X 0,Y 418.256,Z 329.881,A -85,B 0,C 180,E1 -10035.112,E2 -10035.112} C_VEL
LIN {X 0,Y 418.289,Z 329.884,A -85,B 0,C 180,E1 -10037.774,E2 -10037.774} C_VEL
LIN {X 0,Y 418.261,Z 329.885,A -85,B 0,C 180,E1 -10041.56,E2 -10041.56} C_VEL
LIN {X 0,Y 418.256,Z 329.883,A -85,B 0,C 180,E1 -10045.159,E2 -10045.159} C_VEL
LIN {X 0,Y 418.242,Z 329.888,A -85,B 0,C 180,E1 -10047.472,E2 -10047.472} C_VEL
LIN {X 0,Y 418.265,Z 329.881,A -85,B 0,C 180,E1 -10050.896,E2 -10050.896} C_VEL
LIN {X 0,Y 418.268,Z 329.881,A -85,B 0,C 180,E1 -10054.096,E2 -10054.096} C_VEL
LIN {X 0,Y 418.23,Z 329.89,A -85,B 0,C 180,E1 -10057.264,E2 -10057.264} C_VEL
LIN {X 0,Y 418.281,Z 329.878,A -85,B 0,C 180,E1 -10060.365,E2 -10060.365} C_VEL
LIN {X 0,Y 418.315,Z 329.879,A -85,B 0,C 180,E1 -10063.405,E2 -10063.405} C_VEL
LIN {X 0,Y 418.344,Z 329.876,A -85,B 0,C 180,E1 -10067,E2 -10067} C_VEL
LIN {X 0,Y 418.34,Z 329.871,A -85,B 0,C 180,E1 -10070.329,E2 -10070.329} C_VEL
LIN {X 0,Y 418.486,Z 329.857,A -85,B 0,C 180,E1 -10073.249,E2 -10073.249} C_VEL
LIN {X 0,Y 418.338,Z 329.875,A -85,B 0,C 180,E1 -10075.182,E2 -10075.182} C_VEL
LIN {X 0,Y 418.544,Z 329.846,A -85,B 0,C 180,E1 -10078.076,E2 -10078.076} C_VEL
LIN {X 0,Y 418.67,Z 329.83,A -85,B 0,C 180,E1 -10080.001,E2 -10080.001} C_VEL
LIN {X 0,Y 418.508,Z 329.855,A -85,B 0,C 180,E1 -10082.888,E2 -10082.888} C_VEL
LIN {X 0,Y 418.487,Z 329.859,A -85,B 0,C 180,E1 -10086.752,E2 -10086.752} C_VEL
LIN {X 0,Y 418.341,Z 329.871,A -85,B 0,C 180,E1 -10089.672,E2 -10089.672} C_VEL
LIN {X 0,Y 418.346,Z 329.872,A -85,B 0,C 180,E1 -10093.001,E2 -10093.001} C_VEL
LIN {X 0,Y 418.312,Z 329.878,A -85,B 0,C 180,E1 -10096.736,E2 -10096.736} C_VEL
LIN {X 0,Y 418.27,Z 329.881,A -85,B 0,C 180,E1 -10099.791,E2 -10099.791} C_VEL
LIN {X 0,Y 418.232,Z 329.886,A -85,B 0,C 180,E1 -10102.737,E2 -10102.737} C_VEL
LIN {X 0,Y 418.268,Z 329.883,A -85,B 0,C 180,E1 -10105.905,E2 -10105.905} C_VEL
LIN {X 0,Y 418.265,Z 329.88,A -85,B 0,C 180,E1 -10109.162,E2 -10109.162} C_VEL
LIN {X 0,Y 418.258,Z 329.881,A -85,B 0,C 180,E1 -10112.844,E2 -10112.844} C_VEL
LIN {X 0,Y 418.246,Z 329.889,A -85,B 0,C 180,E1 -10116.238,E2 -10116.238} C_VEL
LIN {X 0,Y 418.275,Z 329.966,A -85,B 0,C 180,E1 -10119.68,E2 -10119.68} C_VEL
LIN {X 0,Y 418.645,Z 332.542,A -85,B 0,C 180,E1 -10122.384,E2 -10122.384} C_VEL
LIN {X 0,Y 419.06,Z 335.465,A -85,B 0,C 180,E1 -10125.221,E2 -10125.221} C_VEL
LIN {X 0,Y 419.243,Z 338.458,A -85,B 0,C 180,E1 -10127.891,E2 -10127.891} C_VEL
LIN {X 0,Y 419.083,Z 341.6,A -85,B 0,C 180,E1 -10130.482,E2 -10130.482} C_VEL
LIN {X 0,Y 418.746,Z 346.192,A -85,B 0,C 180,E1 -10134.026,E2 -10134.026} C_VEL
LIN {X 0,Y 418.382,Z 350.945,A -85,B 0,C 180,E1 -10137.484,E2 -10137.484} C_VEL
LIN {X 0,Y 418.001,Z 355.783,A -85,B 0,C 180,E1 -10140.818,E2 -10140.818} C_VEL
LIN {X 0,Y 417.702,Z 360.699,A -85,B 0,C 180,E1 -10144.058,E2 -10144.058} C_VEL
LIN {X 0,Y 417.478,Z 365.67,A -85,B 0,C 180,E1 -10147.22,E2 -10147.22} C_VEL
LIN {X 0,Y 417.255,Z 371.136,A -85,B 0,C 180,E1 -10150.603,E2 -10150.603} C_VEL
LIN {X 0,Y 417.148,Z 374.69,A -85,B 0,C 180,E1 -10152.744,E2 -10152.744} C_VEL
LIN {X 0,Y 419.489,Z 387.07,A -85,B 0,C 180,E1 -10153.232,E2 -10153.232} C_VEL
LIN {X 0,Y 421.312,Z 399.762,A -85,B 0,C 180,E1 -10153.888,E2 -10153.888} C_VEL
LIN {X 0,Y 421.623,Z 402.607,A -85,B 0,C 180,E1 -10154.073,E2 -10154.073} C_VEL
LIN {X 0,Y 420.969,Z 413.152,A -85,B 0,C 180,E1 -10154.755,E2 -10154.755} C_VEL
LIN {X 0,Y 420.396,Z 422.151,A -85,B 0,C 180,E1 -10155.477,E2 -10155.477} C_VEL
LIN {X 0,Y 419.835,Z 430.029,A -85,B 0,C 180,E1 -10156.23,E2 -10156.23} C_VEL
LIN {X 0,Y 419.354,Z 438.281,A -85,B 0,C 180,E1 -10157.17,E2 -10157.17} C_VEL
LIN {X 0,Y 418.812,Z 445.501,A -85,B 0,C 180,E1 -10158.138,E2 -10158.138} C_VEL
LIN {X 0,Y 418.314,Z 451.703,A -85,B 0,C 180,E1 -10159.105,E2 -10159.105} C_VEL
LIN {X 0,Y 417.849,Z 458.24,A -85,B 0,C 180,E1 -10160.317,E2 -10160.317} C_VEL
LIN {X 0,Y 417.649,Z 462.745,A -85,B 0,C 180,E1 -10161.289,E2 -10161.289} C_VEL
LIN {X 0,Y 417.291,Z 468.234,A -85,B 0,C 180,E1 -10162.743,E2 -10162.743} C_VEL
LIN {X 0,Y 417.113,Z 472.558,A -85,B 0,C 180,E1 -10164.198,E2 -10164.198} C_VEL
LIN {X 0,Y 417.11,Z 474.926,A -85,B 0,C 180,E1 -10165.167,E2 -10165.167} C_VEL
LIN {X 0,Y 417.029,Z 478.108,A -85,B 0,C 180,E1 -10167.102,E2 -10167.102} C_VEL
LIN {X 0,Y 417.057,Z 479.166,A -85,B 0,C 180,E1 -10168.069,E2 -10168.069} C_VEL
LIN {X 0,Y 417.011,Z 479.753,A -85,B 0,C 180,E1 -10169.034,E2 -10169.034} C_VEL
LIN {X 0,Y 417.011,Z 479.753,A -85,B 0,C 180,E1 -10170.966,E2 -10170.966} C_VEL
LIN {X 0,Y 417.057,Z 479.166,A -85,B 0,C 180,E1 -10171.931,E2 -10171.931} C_VEL
LIN {X 0,Y 417.016,Z 476.721,A -85,B 0,C 180,E1 -10173.865,E2 -10173.865} C_VEL
LIN {X 0,Y 417.127,Z 473.776,A -85,B 0,C 180,E1 -10175.317,E2 -10175.317} C_VEL
LIN {X 0,Y 417.236,Z 469.788,A -85,B 0,C 180,E1 -10176.771,E2 -10176.771} C_VEL
LIN {X 0,Y 417.491,Z 464.659,A -85,B 0,C 180,E1 -10178.227,E2 -10178.227} C_VEL
LIN {X 0,Y 417.791,Z 459.397,A -85,B 0,C 180,E1 -10179.44,E2 -10179.44} C_VEL
LIN {X 0,Y 418.194,Z 453.078,A -85,B 0,C 180,E1 -10180.653,E2 -10180.653} C_VEL
LIN {X 0,Y 418.661,Z 447.127,A -85,B 0,C 180,E1 -10181.621,E2 -10181.621} C_VEL
LIN {X 0,Y 419.2,Z 440.2,A -85,B 0,C 180,E1 -10182.588,E2 -10182.588} C_VEL
LIN {X 0,Y 419.728,Z 432.017,A -85,B 0,C 180,E1 -10183.557,E2 -10183.557} C_VEL
LIN {X 0,Y 420.289,Z 423.363,A -85,B 0,C 180,E1 -10184.415,E2 -10184.415} C_VEL
LIN {X 0,Y 420.875,Z 414.785,A -85,B 0,C 180,E1 -10185.124,E2 -10185.124} C_VEL
LIN {X 0,Y 421.393,Z 406.335,A -85,B 0,C 180,E1 -10185.706,E2 -10185.706} C_VEL
LIN {X 0,Y 421.465,Z 400.739,A -85,B 0,C 180,E1 -10186.048,E2 -10186.048} C_VEL
LIN {X 0,Y 419.486,Z 387.049,A -85,B 0,C 180,E1 -10186.768,E2 -10186.768} C_VEL
LIN {X 0,Y 417.267,Z 375.727,A -85,B 0,C 180,E1 -10187.219,E2 -10187.219} C_VEL
LIN {X 0,Y 417.134,Z 374.658,A -85,B 0,C 180,E1 -10187.275,E2 -10187.275} C_VEL
LIN {X 0,Y 417.286,Z 370.66,A -85,B 0,C 180,E1 -10189.685,E2 -10189.685} C_VEL
LIN {X 0,Y 417.451,Z 365.635,A -85,B 0,C 180,E1 -10192.781,E2 -10192.781} C_VEL
LIN {X 0,Y 417.635,Z 362.33,A -85,B 0,C 180,E1 -10194.879,E2 -10194.879} C_VEL
LIN {X 0,Y 417.914,Z 357.407,A -85,B 0,C 180,E1 -10198.091,E2 -10198.091} C_VEL
LIN {X 0,Y 418.234,Z 352.539,A -85,B 0,C 180,E1 -10201.394,E2 -10201.394} C_VEL
LIN {X 0,Y 418.578,Z 347.968,A -85,B 0,C 180,E1 -10204.641,E2 -10204.641} C_VEL
LIN {X 0,Y 418.907,Z 343.575,A -85,B 0,C 180,E1 -10207.952,E2 -10207.952} C_VEL
LIN {X 0,Y 419.184,Z 339.737,A -85,B 0,C 180,E1 -10211.021,E2 -10211.021} C_VEL
LIN {X 0,Y 419.183,Z 336.935,A -85,B 0,C 180,E1 -10213.425,E2 -10213.425} C_VEL
LIN {X 0,Y 418.772,Z 333.639,A -85,B 0,C 180,E1 -10216.521,E2 -10216.521} C_VEL
LIN {X 0,Y 418.451,Z 331.098,A -85,B 0,C 180,E1 -10219.094,E2 -10219.094} C_VEL
LIN {X 0,Y 418.267,Z 329.886,A -85,B 0,C 180,E1 -10220.617,E2 -10220.617} C_VEL
LIN {X 0,Y 418.244,Z 329.89,A -85,B 0,C 180,E1 -10223.975,E2 -10223.975} C_VEL
LIN {X 0,Y 418.258,Z 329.881,A -85,B 0,C 180,E1 -10227.156,E2 -10227.156} C_VEL
LIN {X 0,Y 418.269,Z 329.88,A -85,B 0,C 180,E1 -10230.895,E2 -10230.895} C_VEL
LIN {X 0,Y 418.268,Z 329.883,A -85,B 0,C 180,E1 -10234.095,E2 -10234.095} C_VEL
LIN {X 0,Y 418.232,Z 329.886,A -85,B 0,C 180,E1 -10237.263,E2 -10237.263} C_VEL
LIN {X 0,Y 418.283,Z 329.878,A -85,B 0,C 180,E1 -10240.364,E2 -10240.364} C_VEL
LIN {X 0,Y 418.316,Z 329.879,A -85,B 0,C 180,E1 -10243.404,E2 -10243.404} C_VEL
LIN {X 0,Y 418.346,Z 329.872,A -85,B 0,C 180,E1 -10246.999,E2 -10246.999} C_VEL
LIN {X 0,Y 418.341,Z 329.871,A -85,B 0,C 180,E1 -10250.328,E2 -10250.328} C_VEL
LIN {X 0,Y 418.487,Z 329.859,A -85,B 0,C 180,E1 -10253.248,E2 -10253.248} C_VEL
LIN {X 0,Y 418.337,Z 329.877,A -85,B 0,C 180,E1 -10255.181,E2 -10255.181} C_VEL
LIN {X 0,Y 418.543,Z 329.846,A -85,B 0,C 180,E1 -10258.075,E2 -10258.075} C_VEL
LIN {X 0,Y 418.67,Z 329.83,A -85,B 0,C 180,E1 -10259.999,E2 -10259.999} C_VEL
LIN {X 0,Y 418.509,Z 329.854,A -85,B 0,C 180,E1 -10262.887,E2 -10262.887} C_VEL
LIN {X 0,Y 418.486,Z 329.857,A -85,B 0,C 180,E1 -10266.751,E2 -10266.751} C_VEL
LIN {X 0,Y 418.34,Z 329.871,A -85,B 0,C 180,E1 -10269.671,E2 -10269.671} C_VEL
LIN {X 0,Y 418.344,Z 329.876,A -85,B 0,C 180,E1 -10273,E2 -10273} C_VEL
LIN {X 0,Y 418.311,Z 329.881,A -85,B 0,C 180,E1 -10276.735,E2 -10276.735} C_VEL
LIN {X 0,Y 418.269,Z 329.88,A -85,B 0,C 180,E1 -10279.79,E2 -10279.79} C_VEL
LIN {X 0,Y 418.23,Z 329.89,A -85,B 0,C 180,E1 -10282.736,E2 -10282.736} C_VEL
LIN {X 0,Y 418.268,Z 329.881,A -85,B 0,C 180,E1 -10285.904,E2 -10285.904} C_VEL
LIN {X 0,Y 418.262,Z 329.881,A -85,B 0,C 180,E1 -10289.161,E2 -10289.161} C_VEL
LIN {X 0,Y 418.254,Z 329.884,A -85,B 0,C 180,E1 -10292.844,E2 -10292.844} C_VEL
LIN {X 0,Y 418.245,Z 329.889,A -85,B 0,C 180,E1 -10296.238,E2 -10296.238} C_VEL
LIN {X 0,Y 418.262,Z 329.882,A -85,B 0,C 180,E1 -10299.68,E2 -10299.68} C_VEL
LIN {X 0,Y 418.282,Z 329.883,A -85,B 0,C 180,E1 -10302.329,E2 -10302.329} C_VEL
LIN {X 0,Y 418.25,Z 329.882,A -85,B 0,C 180,E1 -10305.111,E2 -10305.111} C_VEL
LIN {X 0,Y 418.253,Z 329.886,A -85,B 0,C 180,E1 -10307.769,E2 -10307.769} C_VEL
LIN {X 0,Y 418.263,Z 329.881,A -85,B 0,C 180,E1 -10310.617,E2 -10310.617} C_VEL
LIN {X 0,Y 418.242,Z 329.889,A -85,B 0,C 180,E1 -10313.976,E2 -10313.976} C_VEL
LIN {X 0,Y 418.254,Z 329.882,A -85,B 0,C 180,E1 -10317.156,E2 -10317.156} C_VEL
LIN {X 0,Y 418.265,Z 329.88,A -85,B 0,C 180,E1 -10320.895,E2 -10320.895} C_VEL
LIN {X 0,Y 418.267,Z 329.882,A -85,B 0,C 180,E1 -10324.096,E2 -10324.096} C_VEL
LIN {X 0,Y 418.234,Z 329.888,A -85,B 0,C 180,E1 -10327.264,E2 -10327.264} C_VEL
LIN {X 0,Y 418.28,Z 329.879,A -85,B 0,C 180,E1 -10330.364,E2 -10330.364} C_VEL
LIN {X 0,Y 418.313,Z 329.882,A -85,B 0,C 180,E1 -10333.405,E2 -10333.405} C_VEL
LIN {X 0,Y 418.343,Z 329.877,A -85,B 0,C 180,E1 -10336.999,E2 -10336.999} C_VEL
LIN {X 0,Y 418.338,Z 329.876,A -85,B 0,C 180,E1 -10340.329,E2 -10340.329} C_VEL
LIN {X 0,Y 418.491,Z 329.857,A -85,B 0,C 180,E1 -10343.249,E2 -10343.249} C_VEL
LIN {X 0,Y 418.338,Z 329.877,A -85,B 0,C 180,E1 -10345.182,E2 -10345.182} C_VEL
LIN {X 0,Y 418.542,Z 329.849,A -85,B 0,C 180,E1 -10348.075,E2 -10348.075} C_VEL
LIN {X 0,Y 418.67,Z 329.835,A -85,B 0,C 180,E1 -10350,E2 -10350} C_VEL
LIN {X 0,Y 418.507,Z 329.855,A -85,B 0,C 180,E1 -10352.888,E2 -10352.888} C_VEL
LIN {X 0,Y 418.491,Z 329.857,A -85,B 0,C 180,E1 -10356.751,E2 -10356.751} C_VEL
LIN {X 0,Y 418.338,Z 329.876,A -85,B 0,C 180,E1 -10359.671,E2 -10359.671} C_VEL
LIN {X 0,Y 418.32,Z 329.878,A -85,B 0,C 180,E1 -10363.319,E2 -10363.319} C_VEL
LIN {X 0,Y 417.626,Z 329.965,A -85,B 0,C 180,E1 -10364.122,E2 -10364.122} C_VEL
LIN {X 0,Y 414.748,Z 330.323,A -85,B 0,C 180,E1 -10365.428,E2 -10365.428} C_VEL
LIN {X 0,Y 412.335,Z 330.625,A -85,B 0,C 180,E1 -10366.482,E2 -10366.482} C_VEL
LIN {X 0,Y 411.313,Z 330.751,A -85,B 0,C 180,E1 -10367.297,E2 -10367.297} C_VEL
LIN {X 0,Y 411.236,Z 330.759,A -85,B 0,C 180,E1 -10367.573,E2 -10367.573} C_VEL
LIN {X 0,Y 411.193,Z 330.763,A -85,B 0,C 180,E1 -10371.034,E2 -10371.034} C_VEL
LIN {X 0,Y 411.224,Z 330.762,A -85,B 0,C 180,E1 -10374.215,E2 -10374.215} C_VEL
LIN {X 0,Y 411.255,Z 330.753,A -85,B 0,C 180,E1 -10377.478,E2 -10377.478} C_VEL
LIN {X 0,Y 411.185,Z 330.763,A -85,B 0,C 180,E1 -10380.848,E2 -10380.848} C_VEL
LIN {X 0,Y 411.203,Z 330.765,A -85,B 0,C 180,E1 -10384.334,E2 -10384.334} C_VEL
LIN {X 0,Y 411.2,Z 330.766,A -85,B 0,C 180,E1 -10387.973,E2 -10387.973} C_VEL
LIN {X 0,Y 411.196,Z 330.761,A -85,B 0,C 180,E1 -10391.234,E2 -10391.234} C_VEL
LIN {X 0,Y 411.183,Z 330.764,A -85,B 0,C 180,E1 -10394.489,E2 -10394.489} C_VEL
LIN {X 0,Y 411.227,Z 330.758,A -85,B 0,C 180,E1 -10397.297,E2 -10397.297} C_VEL
LIN {X 0,Y 411.227,Z 330.757,A -85,B 0,C 180,E1 -10400.778,E2 -10400.778} C_VEL
LIN {X 0,Y 411.196,Z 330.761,A -85,B 0,C 180,E1 -10404.472,E2 -10404.472} C_VEL
LIN {X 0,Y 411.204,Z 330.76,A -85,B 0,C 180,E1 -10406.874,E2 -10406.874} C_VEL
LIN {X 0,Y 411.23,Z 330.757,A -85,B 0,C 180,E1 -10410.645,E2 -10410.645} C_VEL
LIN {X 0,Y 411.235,Z 330.761,A -85,B 0,C 180,E1 -10413.62,E2 -10413.62} C_VEL
LIN {X 0,Y 411.194,Z 330.763,A -85,B 0,C 180,E1 -10416.853,E2 -10416.853} C_VEL
LIN {X 0,Y 411.213,Z 330.759,A -85,B 0,C 180,E1 -10420.051,E2 -10420.051} C_VEL
LIN {X 0,Y 411.261,Z 330.759,A -85,B 0,C 180,E1 -10423.132,E2 -10423.132} C_VEL
LIN {X 0,Y 411.304,Z 330.751,A -85,B 0,C 180,E1 -10426.896,E2 -10426.896} C_VEL
LIN {X 0,Y 411.292,Z 330.749,A -85,B 0,C 180,E1 -10430.162,E2 -10430.162} C_VEL
LIN {X 0,Y 411.45,Z 330.734,A -85,B 0,C 180,E1 -10433.133,E2 -10433.133} C_VEL
LIN {X 0,Y 411.309,Z 330.752,A -85,B 0,C 180,E1 -10435.1,E2 -10435.1} C_VEL
LIN {X 0,Y 411.513,Z 330.721,A -85,B 0,C 180,E1 -10438.043,E2 -10438.043} C_VEL
LIN {X 0,Y 411.639,Z 330.706,A -85,B 0,C 180,E1 -10440.001,E2 -10440.001} C_VEL
LIN {X 0,Y 411.464,Z 330.732,A -85,B 0,C 180,E1 -10442.938,E2 -10442.938} C_VEL
LIN {X 0,Y 411.451,Z 330.733,A -85,B 0,C 180,E1 -10446.868,E2 -10446.868} C_VEL
LIN {X 0,Y 411.293,Z 330.749,A -85,B 0,C 180,E1 -10449.839,E2 -10449.839} C_VEL
LIN {X 0,Y 411.305,Z 330.748,A -85,B 0,C 180,E1 -10453.105,E2 -10453.105} C_VEL
LIN {X 0,Y 411.263,Z 330.754,A -85,B 0,C 180,E1 -10456.869,E2 -10456.869} C_VEL
LIN {X 0,Y 411.231,Z 330.759,A -85,B 0,C 180,E1 -10459.987,E2 -10459.987} C_VEL
LIN {X 0,Y 411.196,Z 330.761,A -85,B 0,C 180,E1 -10463.148,E2 -10463.148} C_VEL
LIN {X 0,Y 411.237,Z 330.76,A -85,B 0,C 180,E1 -10466.381,E2 -10466.381} C_VEL
LIN {X 0,Y 411.201,Z 330.763,A -85,B 0,C 180,E1 -10469.713,E2 -10469.713} C_VEL
LIN {X 0,Y 411.207,Z 330.759,A -85,B 0,C 180,E1 -10473.156,E2 -10473.156} C_VEL
LIN {X 0,Y 411.194,Z 330.766,A -85,B 0,C 180,E1 -10476.553,E2 -10476.553} C_VEL
LIN {X 0,Y 411.229,Z 330.763,A -85,B 0,C 180,E1 -10479.223,E2 -10479.223} C_VEL
LIN {X 0,Y 411.674,Z 334.05,A -85,B 0,C 180,E1 -10482.77,E2 -10482.77} C_VEL
LIN {X 0,Y 412.109,Z 337.106,A -85,B 0,C 180,E1 -10485.747,E2 -10485.747} C_VEL
LIN {X 0,Y 412.165,Z 340.351,A -85,B 0,C 180,E1 -10488.614,E2 -10488.614} C_VEL
LIN {X 0,Y 411.929,Z 344.09,A -85,B 0,C 180,E1 -10491.704,E2 -10491.704} C_VEL
LIN {X 0,Y 411.624,Z 347.724,A -85,B 0,C 180,E1 -10494.514,E2 -10494.514} C_VEL
LIN {X 0,Y 411.241,Z 352.498,A -85,B 0,C 180,E1 -10498.009,E2 -10498.009} C_VEL
LIN {X 0,Y 410.874,Z 357.33,A -85,B 0,C 180,E1 -10501.384,E2 -10501.384} C_VEL
LIN {X 0,Y 410.598,Z 362.245,A -85,B 0,C 180,E1 -10504.665,E2 -10504.665} C_VEL
LIN {X 0,Y 410.356,Z 367.21,A -85,B 0,C 180,E1 -10507.865,E2 -10507.865} C_VEL
LIN {X 0,Y 410.135,Z 372.198,A -85,B 0,C 180,E1 -10510.999,E2 -10510.999} C_VEL
LIN {X 0,Y 410.084,Z 374.47,A -85,B 0,C 180,E1 -10512.419,E2 -10512.419} C_VEL
LIN {X 0,Y 413.111,Z 390.816,A -85,B 0,C 180,E1 -10513.126,E2 -10513.126} C_VEL
LIN {X 0,Y 414.469,Z 401.154,A -85,B 0,C 180,E1 -10513.712,E2 -10513.712} C_VEL
LIN {X 0,Y 414.447,Z 408.124,A -85,B 0,C 180,E1 -10514.148,E2 -10514.148} C_VEL
LIN {X 0,Y 413.587,Z 420.602,A -85,B 0,C 180,E1 -10515.107,E2 -10515.107} C_VEL
LIN {X 0,Y 412.907,Z 429.659,A -85,B 0,C 180,E1 -10515.975,E2 -10515.975} C_VEL
LIN {X 0,Y 412.398,Z 438.084,A -85,B 0,C 180,E1 -10516.95,E2 -10516.95} C_VEL
LIN {X 0,Y 411.824,Z 445.304,A -85,B 0,C 180,E1 -10517.933,E2 -10517.933} C_VEL
LIN {X 0,Y 411.321,Z 451.506,A -85,B 0,C 180,E1 -10518.918,E2 -10518.918} C_VEL
LIN {X 0,Y 410.827,Z 458.044,A -85,B 0,C 180,E1 -10520.15,E2 -10520.15} C_VEL
LIN {X 0,Y 410.587,Z 462.548,A -85,B 0,C 180,E1 -10521.138,E2 -10521.138} C_VEL
LIN {X 0,Y 410.213,Z 468.038,A -85,B 0,C 180,E1 -10522.617,E2 -10522.617} C_VEL
LIN {X 0,Y 410.037,Z 472.362,A -85,B 0,C 180,E1 -10524.097,E2 -10524.097} C_VEL
LIN {X 0,Y 410.023,Z 474.729,A -85,B 0,C 180,E1 -10525.084,E2 -10525.084} C_VEL
LIN {X 0,Y 409.934,Z 476.526,A -85,B 0,C 180,E1 -10526.068,E2 -10526.068} C_VEL
LIN {X 0,Y 409.967,Z 478.971,A -85,B 0,C 180,E1 -10528.035,E2 -10528.035} C_VEL
LIN {X 0,Y 409.936,Z 479.558,A -85,B 0,C 180,E1 -10529.018,E2 -10529.018} C_VEL
LIN {X 0,Y 409.936,Z 479.558,A -85,B 0,C 180,E1 -10530.982,E2 -10530.982} C_VEL
LIN {X 0,Y 409.967,Z 478.971,A -85,B 0,C 180,E1 -10531.965,E2 -10531.965} C_VEL
LIN {X 0,Y 409.934,Z 476.526,A -85,B 0,C 180,E1 -10533.932,E2 -10533.932} C_VEL
LIN {X 0,Y 410.023,Z 473.579,A -85,B 0,C 180,E1 -10535.409,E2 -10535.409} C_VEL
LIN {X 0,Y 410.17,Z 469.592,A -85,B 0,C 180,E1 -10536.889,E2 -10536.889} C_VEL
LIN {X 0,Y 410.451,Z 464.463,A -85,B 0,C 180,E1 -10538.369,E2 -10538.369} C_VEL
LIN {X 0,Y 410.759,Z 459.2,A -85,B 0,C 180,E1 -10539.603,E2 -10539.603} C_VEL
LIN {X 0,Y 411.178,Z 452.881,A -85,B 0,C 180,E1 -10540.837,E2 -10540.837} C_VEL
LIN {X 0,Y 411.681,Z 446.931,A -85,B 0,C 180,E1 -10541.821,E2 -10541.821} C_VEL
LIN {X 0,Y 412.239,Z 440.003,A -85,B 0,C 180,E1 -10542.805,E2 -10542.805} C_VEL
LIN {X 0,Y 412.789,Z 431.82,A -85,B 0,C 180,E1 -10543.79,E2 -10543.79} C_VEL
LIN {X 0,Y 413.383,Z 423.299,A -85,B 0,C 180,E1 -10544.649,E2 -10544.649} C_VEL
LIN {X 0,Y 413.995,Z 414.588,A -85,B 0,C 180,E1 -10545.382,E2 -10545.382} C_VEL
LIN {X 0,Y 414.645,Z 404.646,A -85,B 0,C 180,E1 -10546.062,E2 -10546.062} C_VEL
LIN {X 0,Y 414.046,Z 397.176,A -85,B 0,C 180,E1 -10546.523,E2 -10546.523} C_VEL
LIN {X 0,Y 412.174,Z 385.46,A -85,B 0,C 180,E1 -10547.125,E2 -10547.125} C_VEL
LIN {X 0,Y 410.084,Z 374.47,A -85,B 0,C 180,E1 -10547.581,E2 -10547.581} C_VEL
LIN {X 0,Y 410.208,Z 370.494,A -85,B 0,C 180,E1 -10550.039,E2 -10550.039} C_VEL
LIN {X 0,Y 410.403,Z 365.512,A -85,B 0,C 180,E1 -10553.195,E2 -10553.195} C_VEL
LIN {X 0,Y 410.672,Z 360.585,A -85,B 0,C 180,E1 -10556.42,E2 -10556.42} C_VEL
LIN {X 0,Y 410.983,Z 355.706,A -85,B 0,C 180,E1 -10559.73,E2 -10559.73} C_VEL
LIN {X 0,Y 411.242,Z 352.475,A -85,B 0,C 180,E1 -10561.99,E2 -10561.99} C_VEL
LIN {X 0,Y 411.601,Z 347.702,A -85,B 0,C 180,E1 -10565.489,E2 -10565.489} C_VEL
LIN {X 0,Y 411.916,Z 344.088,A -85,B 0,C 180,E1 -10568.294,E2 -10568.294} C_VEL
LIN {X 0,Y 412.173,Z 339.977,A -85,B 0,C 180,E1 -10571.682,E2 -10571.682} C_VEL
LIN {X 0,Y 412.08,Z 336.983,A -85,B 0,C 180,E1 -10574.367,E2 -10574.367} C_VEL
LIN {X 0,Y 411.53,Z 333.064,A -85,B 0,C 180,E1 -10578.238,E2 -10578.238} C_VEL
LIN {X 0,Y 411.229,Z 330.763,A -85,B 0,C 180,E1 -10580.777,E2 -10580.777} C_VEL
LIN {X 0,Y 411.199,Z 330.769,A -85,B 0,C 180,E1 -10584.471,E2 -10584.471} C_VEL
LIN {X 0,Y 411.208,Z 330.759,A -85,B 0,C 180,E1 -10586.873,E2 -10586.873} C_VEL
LIN {X 0,Y 411.234,Z 330.756,A -85,B 0,C 180,E1 -10590.644,E2 -10590.644} C_VEL
LIN {X 0,Y 411.237,Z 330.76,A -85,B 0,C 180,E1 -10593.619,E2 -10593.619} C_VEL
LIN {X 0,Y 411.196,Z 330.761,A -85,B 0,C 180,E1 -10596.852,E2 -10596.852} C_VEL
LIN {X 0,Y 411.215,Z 330.761,A -85,B 0,C 180,E1 -10600.05,E2 -10600.05} C_VEL
LIN {X 0,Y 411.263,Z 330.754,A -85,B 0,C 180,E1 -10603.131,E2 -10603.131} C_VEL
LIN {X 0,Y 411.305,Z 330.748,A -85,B 0,C 180,E1 -10606.895,E2 -10606.895} C_VEL
LIN {X 0,Y 411.293,Z 330.749,A -85,B 0,C 180,E1 -10610.161,E2 -10610.161} C_VEL
LIN {X 0,Y 411.451,Z 330.733,A -85,B 0,C 180,E1 -10613.132,E2 -10613.132} C_VEL
LIN {X 0,Y 411.309,Z 330.751,A -85,B 0,C 180,E1 -10615.098,E2 -10615.098} C_VEL
LIN {X 0,Y 411.512,Z 330.721,A -85,B 0,C 180,E1 -10618.042,E2 -10618.042} C_VEL
LIN {X 0,Y 411.639,Z 330.706,A -85,B 0,C 180,E1 -10619.999,E2 -10619.999} C_VEL
LIN {X 0,Y 411.464,Z 330.732,A -85,B 0,C 180,E1 -10622.937,E2 -10622.937} C_VEL
LIN {X 0,Y 411.45,Z 330.734,A -85,B 0,C 180,E1 -10626.867,E2 -10626.867} C_VEL
LIN {X 0,Y 411.292,Z 330.749,A -85,B 0,C 180,E1 -10629.838,E2 -10629.838} C_VEL
LIN {X 0,Y 411.304,Z 330.751,A -85,B 0,C 180,E1 -10633.104,E2 -10633.104} C_VEL
LIN {X 0,Y 411.255,Z 330.759,A -85,B 0,C 180,E1 -10636.888,E2 -10636.888} C_VEL
LIN {X 0,Y 411.228,Z 330.757,A -85,B 0,C 180,E1 -10639.986,E2 -10639.986} C_VEL
LIN {X 0,Y 411.194,Z 330.763,A -85,B 0,C 180,E1 -10643.147,E2 -10643.147} C_VEL
LIN {X 0,Y 411.235,Z 330.761,A -85,B 0,C 180,E1 -10646.38,E2 -10646.38} C_VEL
LIN {X 0,Y 411.197,Z 330.761,A -85,B 0,C 180,E1 -10649.712,E2 -10649.712} C_VEL
LIN {X 0,Y 411.203,Z 330.76,A -85,B 0,C 180,E1 -10653.155,E2 -10653.155} C_VEL
LIN {X 0,Y 411.192,Z 330.765,A -85,B 0,C 180,E1 -10656.553,E2 -10656.553} C_VEL
LIN {X 0,Y 411.224,Z 330.759,A -85,B 0,C 180,E1 -10659.73,E2 -10659.73} C_VEL
LIN {X 0,Y 411.221,Z 330.758,A -85,B 0,C 180,E1 -10663.126,E2 -10663.126} C_VEL
LIN {X 0,Y 411.17,Z 330.769,A -85,B 0,C 180,E1 -10665.88,E2 -10665.88} C_VEL
LIN {X 0,Y 411.208,Z 330.761,A -85,B 0,C 180,E1 -10669.499,E2 -10669.499} C_VEL
LIN {X 0,Y 411.2,Z 330.766,A -85,B 0,C 180,E1 -10672.027,E2 -10672.027} C_VEL
LIN {X 0,Y 411.203,Z 330.765,A -85,B 0,C 180,E1 -10675.666,E2 -10675.666} C_VEL
LIN {X 0,Y 411.185,Z 330.763,A -85,B 0,C 180,E1 -10679.152,E2 -10679.152} C_VEL
LIN {X 0,Y 411.255,Z 330.753,A -85,B 0,C 180,E1 -10682.522,E2 -10682.522} C_VEL
LIN {X 0,Y 411.224,Z 330.762,A -85,B 0,C 180,E1 -10685.785,E2 -10685.785} C_VEL
LIN {X 0,Y 411.193,Z 330.763,A -85,B 0,C 180,E1 -10688.966,E2 -10688.966} C_VEL
LIN {X 0,Y 411.249,Z 330.759,A -85,B 0,C 180,E1 -10692.085,E2 -10692.085} C_VEL
LIN {X 0,Y 411.257,Z 330.759,A -85,B 0,C 180,E1 -10695.147,E2 -10695.147} C_VEL
LIN {X 0,Y 411.281,Z 330.753,A -85,B 0,C 180,E1 -10698.167,E2 -10698.167} C_VEL
LIN {X 0,Y 411.478,Z 330.73,A -85,B 0,C 180,E1 -10702.147,E2 -10702.147} C_VEL
LIN {X 0,Y 411.473,Z 330.731,A -85,B 0,C 180,E1 -10704.118,E2 -10704.118} C_VEL
LIN {X 0,Y 411.511,Z 330.725,A -85,B 0,C 180,E1 -10708.043,E2 -10708.043} C_VEL
LIN {X 0,Y 411.639,Z 330.711,A -85,B 0,C 180,E1 -10710,E2 -10710} C_VEL
LIN {X 0,Y 411.463,Z 330.733,A -85,B 0,C 180,E1 -10712.937,E2 -10712.937} C_VEL
LIN {X 0,Y 411.458,Z 330.733,A -85,B 0,C 180,E1 -10716.867,E2 -10716.867} C_VEL
LIN {X 0,Y 411.29,Z 330.754,A -85,B 0,C 180,E1 -10719.839,E2 -10719.839} C_VEL
LIN {X 0,Y 411.281,Z 330.755,A -85,B 0,C 180,E1 -10723.307,E2 -10723.307} C_VEL
LIN {X 0,Y 411.253,Z 330.76,A -85,B 0,C 180,E1 -10726.889,E2 -10726.889} C_VEL
LIN {X 0,Y 411.236,Z 330.759,A -85,B 0,C 180,E1 -10727.573,E2 -10727.573} C_VEL
LIN {X 0,Y 410.575,Z 330.845,A -85,B 0,C 180,E1 -10728.391,E2 -10728.391} C_VEL
LIN {X 0,Y 407.688,Z 331.199,A -85,B 0,C 180,E1 -10729.719,E2 -10729.719} C_VEL
LIN {X 0,Y 405.245,Z 331.506,A -85,B 0,C 180,E1 -10730.792,E2 -10730.792} C_VEL
LIN {X 0,Y 404.208,Z 331.631,A -85,B 0,C 180,E1 -10731.623,E2 -10731.623} C_VEL
LIN {X 0,Y 404.132,Z 331.642,A -85,B 0,C 180,E1 -10731.904,E2 -10731.904} C_VEL
LIN {X 0,Y 404.212,Z 331.631,A -85,B 0,C 180,E1 -10735.297,E2 -10735.297} C_VEL
LIN {X 0,Y 404.192,Z 331.637,A -85,B 0,C 180,E1 -10738,E2 -10738} C_VEL
LIN {X 0,Y 404.135,Z 331.641,A -85,B 0,C 180,E1 -10741.558,E2 -10741.558} C_VEL
LIN {X 0,Y 404.182,Z 331.635,A -85,B 0,C 180,E1 -10745.016,E2 -10745.016} C_VEL
LIN {X 0,Y 404.159,Z 331.638,A -85,B 0,C 180,E1 -10748.756,E2 -10748.756} C_VEL
LIN {X 0,Y 404.146,Z 331.642,A -85,B 0,C 180,E1 -10751.604,E2 -10751.604} C_VEL
LIN {X 0,Y 404.151,Z 331.639,A -85,B 0,C 180,E1 -10754.524,E2 -10754.524} C_VEL
LIN {X 0,Y 404.205,Z 331.633,A -85,B 0,C 180,E1 -10757.305,E2 -10757.305} C_VEL
LIN {X 0,Y 404.165,Z 331.642,A -85,B 0,C 180,E1 -10759.956,E2 -10759.956} C_VEL
LIN {X 0,Y 404.137,Z 331.641,A -85,B 0,C 180,E1 -10763.125,E2 -10763.125} C_VEL
LIN {X 0,Y 404.142,Z 331.641,A -85,B 0,C 180,E1 -10766.188,E2 -10766.188} C_VEL
LIN {X 0,Y 404.142,Z 331.644,A -85,B 0,C 180,E1 -10769.715,E2 -10769.715} C_VEL
LIN {X 0,Y 404.193,Z 331.636,A -85,B 0,C 180,E1 -10773.123,E2 -10773.123} C_VEL
LIN {X 0,Y 404.172,Z 331.642,A -85,B 0,C 180,E1 -10775.335,E2 -10775.335} C_VEL
LIN {X 0,Y 404.136,Z 331.641,A -85,B 0,C 180,E1 -10778.581,E2 -10778.581} C_VEL
LIN {X 0,Y 404.208,Z 331.633,A -85,B 0,C 180,E1 -10781.762,E2 -10781.762} C_VEL
LIN {X 0,Y 404.204,Z 331.635,A -85,B 0,C 180,E1 -10784.883,E2 -10784.883} C_VEL
LIN {X 0,Y 404.255,Z 331.626,A -85,B 0,C 180,E1 -10787.959,E2 -10787.959} C_VEL
LIN {X 0,Y 404.403,Z 331.607,A -85,B 0,C 180,E1 -10792.13,E2 -10792.13} C_VEL
LIN {X 0,Y 404.418,Z 331.605,A -85,B 0,C 180,E1 -10794.016,E2 -10794.016} C_VEL
LIN {X 0,Y 404.482,Z 331.597,A -85,B 0,C 180,E1 -10798.009,E2 -10798.009} C_VEL
LIN {X 0,Y 404.609,Z 331.581,A -85,B 0,C 180,E1 -10800.001,E2 -10800.001} C_VEL
LIN {X 0,Y 404.421,Z 331.609,A -85,B 0,C 180,E1 -10802.989,E2 -10802.989} C_VEL
LIN {X 0,Y 404.399,Z 331.611,A -85,B 0,C 180,E1 -10806.988,E2 -10806.988} C_VEL
LIN {X 0,Y 404.258,Z 331.626,A -85,B 0,C 180,E1 -10810.012,E2 -10810.012} C_VEL
LIN {X 0,Y 404.266,Z 331.625,A -85,B 0,C 180,E1 -10813.212,E2 -10813.212} C_VEL
LIN {X 0,Y 404.216,Z 331.631,A -85,B 0,C 180,E1 -10817.007,E2 -10817.007} C_VEL
LIN {X 0,Y 404.187,Z 331.641,A -85,B 0,C 180,E1 -10820.351,E2 -10820.351} C_VEL
LIN {X 0,Y 404.163,Z 331.637,A -85,B 0,C 180,E1 -10823.575,E2 -10823.575} C_VEL
LIN {X 0,Y 404.183,Z 331.637,A -85,B 0,C 180,E1 -10825.767,E2 -10825.767} C_VEL
LIN {X 0,Y 404.196,Z 331.638,A -85,B 0,C 180,E1 -10828,E2 -10828} C_VEL
LIN {X 0,Y 404.14,Z 331.641,A -85,B 0,C 180,E1 -10831.558,E2 -10831.558} C_VEL
LIN {X 0,Y 404.185,Z 331.636,A -85,B 0,C 180,E1 -10835.017,E2 -10835.017} C_VEL
LIN {X 0,Y 404.16,Z 331.644,A -85,B 0,C 180,E1 -10838.757,E2 -10838.757} C_VEL
LIN {X 0,Y 404.528,Z 334.106,A -85,B 0,C 180,E1 -10841.665,E2 -10841.665} C_VEL
LIN {X 0,Y 405.015,Z 337.768,A -85,B 0,C 180,E1 -10845.354,E2 -10845.354} C_VEL
LIN {X 0,Y 405.152,Z 340.923,A -85,B 0,C 180,E1 -10848.237,E2 -10848.237} C_VEL
LIN {X 0,Y 404.914,Z 344.619,A -85,B 0,C 180,E1 -10851.358,E2 -10851.358} C_VEL
LIN {X 0,Y 404.658,Z 347.694,A -85,B 0,C 180,E1 -10853.807,E2 -10853.807} C_VEL
LIN {X 0,Y 404.258,Z 352.438,A -85,B 0,C 180,E1 -10857.389,E2 -10857.389} C_VEL
LIN {X 0,Y 403.866,Z 357.253,A -85,B 0,C 180,E1 -10860.84,E2 -10860.84} C_VEL
LIN {X 0,Y 403.562,Z 362.128,A -85,B 0,C 180,E1 -10864.191,E2 -10864.191} C_VEL
LIN {X 0,Y 403.302,Z 367.069,A -85,B 0,C 180,E1 -10867.457,E2 -10867.457} C_VEL
LIN {X 0,Y 403.086,Z 372.045,A -85,B 0,C 180,E1 -10870.654,E2 -10870.654} C_VEL
LIN {X 0,Y 403.007,Z 374.318,A -85,B 0,C 180,E1 -10872.124,E2 -10872.124} C_VEL
LIN {X 0,Y 405.146,Z 385.303,A -85,B 0,C 180,E1 -10872.57,E2 -10872.57} C_VEL
LIN {X 0,Y 406.883,Z 395.824,A -85,B 0,C 180,E1 -10873.12,E2 -10873.12} C_VEL
LIN {X 0,Y 407.757,Z 404.765,A -85,B 0,C 180,E1 -10873.679,E2 -10873.679} C_VEL
LIN {X 0,Y 407.142,Z 414.392,A -85,B 0,C 180,E1 -10874.353,E2 -10874.353} C_VEL
LIN {X 0,Y 406.408,Z 424.465,A -85,B 0,C 180,E1 -10875.223,E2 -10875.223} C_VEL
LIN {X 0,Y 405.552,Z 435.968,A -85,B 0,C 180,E1 -10876.471,E2 -10876.471} C_VEL
LIN {X 0,Y 404.841,Z 445.107,A -85,B 0,C 180,E1 -10877.722,E2 -10877.722} C_VEL
LIN {X 0,Y 404.323,Z 451.309,A -85,B 0,C 180,E1 -10878.723,E2 -10878.723} C_VEL
LIN {X 0,Y 403.821,Z 457.848,A -85,B 0,C 180,E1 -10879.977,E2 -10879.977} C_VEL
LIN {X 0,Y 403.546,Z 462.351,A -85,B 0,C 180,E1 -10880.982,E2 -10880.982} C_VEL
LIN {X 0,Y 403.16,Z 467.841,A -85,B 0,C 180,E1 -10882.488,E2 -10882.488} C_VEL
LIN {X 0,Y 402.948,Z 472.165,A -85,B 0,C 180,E1 -10883.993,E2 -10883.993} C_VEL
LIN {X 0,Y 402.935,Z 474.533,A -85,B 0,C 180,E1 -10884.997,E2 -10884.997} C_VEL
LIN {X 0,Y 402.854,Z 476.33,A -85,B 0,C 180,E1 -10885.999,E2 -10885.999} C_VEL
LIN {X 0,Y 402.865,Z 478.775,A -85,B 0,C 180,E1 -10888.001,E2 -10888.001} C_VEL
LIN {X 0,Y 402.863,Z 479.363,A -85,B 0,C 180,E1 -10889,E2 -10889} C_VEL
LIN {X 0,Y 402.863,Z 479.363,A -85,B 0,C 180,E1 -10891,E2 -10891} C_VEL
LIN {X 0,Y 402.865,Z 478.775,A -85,B 0,C 180,E1 -10891.999,E2 -10891.999} C_VEL
LIN {X 0,Y 402.854,Z 476.33,A -85,B 0,C 180,E1 -10894.001,E2 -10894.001} C_VEL
LIN {X 0,Y 402.92,Z 473.382,A -85,B 0,C 180,E1 -10895.505,E2 -10895.505} C_VEL
LIN {X 0,Y 403.083,Z 469.395,A -85,B 0,C 180,E1 -10897.01,E2 -10897.01} C_VEL
LIN {X 0,Y 403.392,Z 464.266,A -85,B 0,C 180,E1 -10898.516,E2 -10898.516} C_VEL
LIN {X 0,Y 403.719,Z 459.003,A -85,B 0,C 180,E1 -10899.772,E2 -10899.772} C_VEL
LIN {X 0,Y 404.173,Z 452.685,A -85,B 0,C 180,E1 -10901.027,E2 -10901.027} C_VEL
LIN {X 0,Y 404.702,Z 446.734,A -85,B 0,C 180,E1 -10902.028,E2 -10902.028} C_VEL
LIN {X 0,Y 405.268,Z 439.806,A -85,B 0,C 180,E1 -10903.029,E2 -10903.029} C_VEL
LIN {X 0,Y 405.855,Z 431.623,A -85,B 0,C 180,E1 -10904.03,E2 -10904.03} C_VEL
LIN {X 0,Y 406.468,Z 423.244,A -85,B 0,C 180,E1 -10904.891,E2 -10904.891} C_VEL
LIN {X 0,Y 407.131,Z 414.392,A -85,B 0,C 180,E1 -10905.648,E2 -10905.648} C_VEL
LIN {X 0,Y 407.776,Z 404.775,A -85,B 0,C 180,E1 -10906.319,E2 -10906.319} C_VEL
LIN {X 0,Y 406.85,Z 395.854,A -85,B 0,C 180,E1 -10906.88,E2 -10906.88} C_VEL
LIN {X 0,Y 405.082,Z 384.924,A -85,B 0,C 180,E1 -10907.447,E2 -10907.447} C_VEL
LIN {X 0,Y 402.999,Z 374.284,A -85,B 0,C 180,E1 -10907.897,E2 -10907.897} C_VEL
LIN {X 0,Y 403.135,Z 370.344,A -85,B 0,C 180,E1 -10910.406,E2 -10910.406} C_VEL
LIN {X 0,Y 403.349,Z 365.397,A -85,B 0,C 180,E1 -10913.625,E2 -10913.625} C_VEL
LIN {X 0,Y 403.672,Z 360.493,A -85,B 0,C 180,E1 -10916.915,E2 -10916.915} C_VEL
LIN {X 0,Y 403.999,Z 355.628,A -85,B 0,C 180,E1 -10920.297,E2 -10920.297} C_VEL
LIN {X 0,Y 404.358,Z 351.278,A -85,B 0,C 180,E1 -10923.459,E2 -10923.459} C_VEL
LIN {X 0,Y 404.72,Z 346.673,A -85,B 0,C 180,E1 -10926.984,E2 -10926.984} C_VEL
LIN {X 0,Y 405.044,Z 342.683,A -85,B 0,C 180,E1 -10930.23,E2 -10930.23} C_VEL
LIN {X 0,Y 405.148,Z 339.998,A -85,B 0,C 180,E1 -10932.572,E2 -10932.572} C_VEL
LIN {X 0,Y 404.893,Z 337.01,A -85,B 0,C 180,E1 -10935.37,E2 -10935.37} C_VEL
LIN {X 0,Y 404.489,Z 333.776,A -85,B 0,C 180,E1 -10938.68,E2 -10938.68} C_VEL
LIN {X 0,Y 404.16,Z 331.643,A -85,B 0,C 180,E1 -10941.243,E2 -10941.243} C_VEL
LIN {X 0,Y 404.185,Z 331.64,A -85,B 0,C 180,E1 -10944.983,E2 -10944.983} C_VEL
LIN {X 0,Y 404.143,Z 331.64,A -85,B 0,C 180,E1 -10948.553,E2 -10948.553} C_VEL
LIN {X 0,Y 404.196,Z 331.638,A -85,B 0,C 180,E1 -10952,E2 -10952} C_VEL
LIN {X 0,Y 404.174,Z 331.638,A -85,B 0,C 180,E1 -10955.334,E2 -10955.334} C_VEL
LIN {X 0,Y 404.138,Z 331.64,A -85,B 0,C 180,E1 -10958.58,E2 -10958.58} C_VEL
LIN {X 0,Y 404.205,Z 331.637,A -85,B 0,C 180,E1 -10961.761,E2 -10961.761} C_VEL
LIN {X 0,Y 404.207,Z 331.632,A -85,B 0,C 180,E1 -10964.882,E2 -10964.882} C_VEL
LIN {X 0,Y 404.256,Z 331.627,A -85,B 0,C 180,E1 -10967.958,E2 -10967.958} C_VEL
LIN {X 0,Y 404.404,Z 331.607,A -85,B 0,C 180,E1 -10972.129,E2 -10972.129} C_VEL
LIN {X 0,Y 404.419,Z 331.606,A -85,B 0,C 180,E1 -10974.014,E2 -10974.014} C_VEL
LIN {X 0,Y 404.481,Z 331.597,A -85,B 0,C 180,E1 -10978.008,E2 -10978.008} C_VEL
LIN {X 0,Y 404.609,Z 331.581,A -85,B 0,C 180,E1 -10979.999,E2 -10979.999} C_VEL
LIN {X 0,Y 404.421,Z 331.61,A -85,B 0,C 180,E1 -10982.988,E2 -10982.988} C_VEL
LIN {X 0,Y 404.398,Z 331.615,A -85,B 0,C 180,E1 -10986.987,E2 -10986.987} C_VEL
LIN {X 0,Y 404.257,Z 331.625,A -85,B 0,C 180,E1 -10990.011,E2 -10990.011} C_VEL
LIN {X 0,Y 404.265,Z 331.627,A -85,B 0,C 180,E1 -10993.211,E2 -10993.211} C_VEL
LIN {X 0,Y 404.214,Z 331.635,A -85,B 0,C 180,E1 -10997.007,E2 -10997.007} C_VEL
LIN {X 0,Y 404.161,Z 331.64,A -85,B 0,C 180,E1 -11000.351,E2 -11000.351} C_VEL
LIN {X 0,Y 404.161,Z 331.637,A -85,B 0,C 180,E1 -11003.574,E2 -11003.574} C_VEL
LIN {X 0,Y 404.181,Z 331.635,A -85,B 0,C 180,E1 -11005.766,E2 -11005.766} C_VEL
LIN {X 0,Y 404.193,Z 331.635,A -85,B 0,C 180,E1 -11007.999,E2 -11007.999} C_VEL
LIN {X 0,Y 404.136,Z 331.64,A -85,B 0,C 180,E1 -11011.558,E2 -11011.558} C_VEL
LIN {X 0,Y 404.182,Z 331.635,A -85,B 0,C 180,E1 -11015.016,E2 -11015.016} C_VEL
LIN {X 0,Y 404.159,Z 331.639,A -85,B 0,C 180,E1 -11018.756,E2 -11018.756} C_VEL
LIN {X 0,Y 404.188,Z 331.635,A -85,B 0,C 180,E1 -11021.61,E2 -11021.61} C_VEL
LIN {X 0,Y 404.188,Z 331.636,A -85,B 0,C 180,E1 -11024.529,E2 -11024.529} C_VEL
LIN {X 0,Y 404.168,Z 331.637,A -85,B 0,C 180,E1 -11027.3,E2 -11027.3} C_VEL
LIN {X 0,Y 404.165,Z 331.644,A -85,B 0,C 180,E1 -11029.955,E2 -11029.955} C_VEL
LIN {X 0,Y 404.137,Z 331.64,A -85,B 0,C 180,E1 -11033.124,E2 -11033.124} C_VEL
LIN {X 0,Y 404.141,Z 331.642,A -85,B 0,C 180,E1 -11036.188,E2 -11036.188} C_VEL
LIN {X 0,Y 404.142,Z 331.646,A -85,B 0,C 180,E1 -11039.715,E2 -11039.715} C_VEL
LIN {X 0,Y 404.191,Z 331.635,A -85,B 0,C 180,E1 -11043.123,E2 -11043.123} C_VEL
LIN {X 0,Y 404.174,Z 331.639,A -85,B 0,C 180,E1 -11045.334,E2 -11045.334} C_VEL
LIN {X 0,Y 404.135,Z 331.64,A -85,B 0,C 180,E1 -11048.581,E2 -11048.581} C_VEL
LIN {X 0,Y 404.207,Z 331.637,A -85,B 0,C 180,E1 -11051.762,E2 -11051.762} C_VEL
LIN {X 0,Y 404.203,Z 331.638,A -85,B 0,C 180,E1 -11054.882,E2 -11054.882} C_VEL
LIN {X 0,Y 404.253,Z 331.628,A -85,B 0,C 180,E1 -11057.958,E2 -11057.958} C_VEL
LIN {X 0,Y 404.43,Z 331.608,A -85,B 0,C 180,E1 -11062.1,E2 -11062.1} C_VEL
LIN {X 0,Y 404.421,Z 331.609,A -85,B 0,C 180,E1 -11064.015,E2 -11064.015} C_VEL
LIN {X 0,Y 404.48,Z 331.601,A -85,B 0,C 180,E1 -11068.009,E2 -11068.009} C_VEL
LIN {X 0,Y 404.608,Z 331.587,A -85,B 0,C 180,E1 -11070,E2 -11070} C_VEL
LIN {X 0,Y 404.42,Z 331.61,A -85,B 0,C 180,E1 -11072.988,E2 -11072.988} C_VEL
LIN {X 0,Y 404.409,Z 331.611,A -85,B 0,C 180,E1 -11076.987,E2 -11076.987} C_VEL
LIN {X 0,Y 404.255,Z 331.631,A -85,B 0,C 180,E1 -11080.012,E2 -11080.012} C_VEL
LIN {X 0,Y 404.263,Z 331.63,A -85,B 0,C 180,E1 -11083.211,E2 -11083.211} C_VEL
LIN {X 0,Y 404.212,Z 331.637,A -85,B 0,C 180,E1 -11087.007,E2 -11087.007} C_VEL
LIN {X 0,Y 404.183,Z 331.64,A -85,B 0,C 180,E1 -11090.35,E2 -11090.35} C_VEL
LIN {X 0,Y 404.132,Z 331.642,A -85,B 0,C 180,E1 -11091.904,E2 -11091.904} C_VEL
LIN {X 0,Y 403.489,Z 331.728,A -85,B 0,C 180,E1 -11092.735,E2 -11092.735} C_VEL
LIN {X 0,Y 400.658,Z 332.088,A -85,B 0,C 180,E1 -11094.087,E2 -11094.087} C_VEL
LIN {X 0,Y 398.249,Z 332.388,A -85,B 0,C 180,E1 -11095.179,E2 -11095.179} C_VEL
LIN {X 0,Y 397.214,Z 332.511,A -85,B 0,C 180,E1 -11096.024,E2 -11096.024} C_VEL
LIN {X 0,Y 397.131,Z 332.518,A -85,B 0,C 180,E1 -11096.31,E2 -11096.31} C_VEL
LIN {X 0,Y 397.119,Z 332.519,A -85,B 0,C 180,E1 -11098.544,E2 -11098.544} C_VEL
LIN {X 0,Y 397.075,Z 332.525,A -85,B 0,C 180,E1 -11102.072,E2 -11102.072} C_VEL
LIN {X 0,Y 397.116,Z 332.516,A -85,B 0,C 180,E1 -11105.504,E2 -11105.504} C_VEL
LIN {X 0,Y 397.133,Z 332.513,A -85,B 0,C 180,E1 -11108.863,E2 -11108.863} C_VEL
LIN {X 0,Y 397.11,Z 332.519,A -85,B 0,C 180,E1 -11112.261,E2 -11112.261} C_VEL
LIN {X 0,Y 397.114,Z 332.515,A -85,B 0,C 180,E1 -11115.065,E2 -11115.065} C_VEL
LIN {X 0,Y 397.152,Z 332.515,A -85,B 0,C 180,E1 -11118.007,E2 -11118.007} C_VEL
LIN {X 0,Y 397.106,Z 332.523,A -85,B 0,C 180,E1 -11121.726,E2 -11121.726} C_VEL
LIN {X 0,Y 397.122,Z 332.519,A -85,B 0,C 180,E1 -11125.507,E2 -11125.507} C_VEL
LIN {X 0,Y 397.075,Z 332.522,A -85,B 0,C 180,E1 -11129.118,E2 -11129.118} C_VEL
LIN {X 0,Y 397.191,Z 332.505,A -85,B 0,C 180,E1 -11132.61,E2 -11132.61} C_VEL
LIN {X 0,Y 397.127,Z 332.515,A -85,B 0,C 180,E1 -11135.982,E2 -11135.982} C_VEL
LIN {X 0,Y 397.136,Z 332.515,A -85,B 0,C 180,E1 -11139.705,E2 -11139.705} C_VEL
LIN {X 0,Y 397.18,Z 332.509,A -85,B 0,C 180,E1 -11142.845,E2 -11142.845} C_VEL
LIN {X 0,Y 397.227,Z 332.503,A -85,B 0,C 180,E1 -11146.703,E2 -11146.703} C_VEL
LIN {X 0,Y 397.216,Z 332.503,A -85,B 0,C 180,E1 -11149.81,E2 -11149.81} C_VEL
LIN {X 0,Y 397.348,Z 332.491,A -85,B 0,C 180,E1 -11152.888,E2 -11152.888} C_VEL
LIN {X 0,Y 397.252,Z 332.505,A -85,B 0,C 180,E1 -11154.926,E2 -11154.926} C_VEL
LIN {X 0,Y 397.451,Z 332.473,A -85,B 0,C 180,E1 -11157.974,E2 -11157.974} C_VEL
LIN {X 0,Y 397.578,Z 332.457,A -85,B 0,C 180,E1 -11160.001,E2 -11160.001} C_VEL
LIN {X 0,Y 397.379,Z 332.485,A -85,B 0,C 180,E1 -11163.042,E2 -11163.042} C_VEL
LIN {X 0,Y 397.37,Z 332.484,A -85,B 0,C 180,E1 -11166.092,E2 -11166.092} C_VEL
LIN {X 0,Y 397.253,Z 332.499,A -85,B 0,C 180,E1 -11169.162,E2 -11169.162} C_VEL
LIN {X 0,Y 397.219,Z 332.506,A -85,B 0,C 180,E1 -11172.259,E2 -11172.259} C_VEL
LIN {X 0,Y 397.179,Z 332.507,A -85,B 0,C 180,E1 -11175.393,E2 -11175.393} C_VEL
LIN {X 0,Y 397.158,Z 332.514,A -85,B 0,C 180,E1 -11178.574,E2 -11178.574} C_VEL
LIN {X 0,Y 397.096,Z 332.519,A -85,B 0,C 180,E1 -11181.819,E2 -11181.819} C_VEL
LIN {X 0,Y 397.153,Z 332.511,A -85,B 0,C 180,E1 -11185.513,E2 -11185.513} C_VEL
LIN {X 0,Y 397.123,Z 332.516,A -85,B 0,C 180,E1 -11188.544,E2 -11188.544} C_VEL
LIN {X 0,Y 397.08,Z 332.526,A -85,B 0,C 180,E1 -11192.072,E2 -11192.072} C_VEL
LIN {X 0,Y 397.12,Z 332.516,A -85,B 0,C 180,E1 -11195.504,E2 -11195.504} C_VEL
LIN {X 0,Y 397.14,Z 332.744,A -85,B 0,C 180,E1 -11198.863,E2 -11198.863} C_VEL
LIN {X 0,Y 397.593,Z 335.735,A -85,B 0,C 180,E1 -11202.199,E2 -11202.199} C_VEL
LIN {X 0,Y 397.94,Z 338.524,A -85,B 0,C 180,E1 -11205.054,E2 -11205.054} C_VEL
LIN {X 0,Y 398.127,Z 341.516,A -85,B 0,C 180,E1 -11207.871,E2 -11207.871} C_VEL
LIN {X 0,Y 397.913,Z 345.149,A -85,B 0,C 180,E1 -11211,E2 -11211} C_VEL
LIN {X 0,Y 397.701,Z 347.666,A -85,B 0,C 180,E1 -11213.071,E2 -11213.071} C_VEL
LIN {X 0,Y 397.268,Z 352.371,A -85,B 0,C 180,E1 -11216.742,E2 -11216.742} C_VEL
LIN {X 0,Y 397.008,Z 355.559,A -85,B 0,C 180,E1 -11219.112,E2 -11219.112} C_VEL
LIN {X 0,Y 396.653,Z 360.401,A -85,B 0,C 180,E1 -11222.569,E2 -11222.569} C_VEL
LIN {X 0,Y 396.303,Z 365.283,A -85,B 0,C 180,E1 -11225.928,E2 -11225.928} C_VEL
LIN {X 0,Y 396.064,Z 370.235,A -85,B 0,C 180,E1 -11229.213,E2 -11229.213} C_VEL
LIN {X 0,Y 395.903,Z 374.131,A -85,B 0,C 180,E1 -11231.795,E2 -11231.795} C_VEL
LIN {X 0,Y 398.027,Z 384.742,A -85,B 0,C 180,E1 -11232.234,E2 -11232.234} C_VEL
LIN {X 0,Y 399.701,Z 394.598,A -85,B 0,C 180,E1 -11232.755,E2 -11232.755} C_VEL
LIN {X 0,Y 400.761,Z 403.321,A -85,B 0,C 180,E1 -11233.305,E2 -11233.305} C_VEL
LIN {X 0,Y 400.565,Z 410.932,A -85,B 0,C 180,E1 -11233.828,E2 -11233.828} C_VEL
LIN {X 0,Y 399.868,Z 420.21,A -85,B 0,C 180,E1 -11234.584,E2 -11234.584} C_VEL
LIN {X 0,Y 399.106,Z 429.16,A -85,B 0,C 180,E1 -11235.468,E2 -11235.468} C_VEL
LIN {X 0,Y 398.579,Z 436.145,A -85,B 0,C 180,E1 -11236.28,E2 -11236.28} C_VEL
LIN {X 0,Y 397.882,Z 444.91,A -85,B 0,C 180,E1 -11237.504,E2 -11237.504} C_VEL
LIN {X 0,Y 397.306,Z 451.112,A -85,B 0,C 180,E1 -11238.521,E2 -11238.521} C_VEL
LIN {X 0,Y 396.804,Z 457.651,A -85,B 0,C 180,E1 -11239.798,E2 -11239.798} C_VEL
LIN {X 0,Y 396.501,Z 462.154,A -85,B 0,C 180,E1 -11240.821,E2 -11240.821} C_VEL
LIN {X 0,Y 396.091,Z 467.645,A -85,B 0,C 180,E1 -11242.353,E2 -11242.353} C_VEL
LIN {X 0,Y 395.863,Z 471.969,A -85,B 0,C 180,E1 -11243.885,E2 -11243.885} C_VEL
LIN {X 0,Y 395.848,Z 474.337,A -85,B 0,C 180,E1 -11244.907,E2 -11244.907} C_VEL
LIN {X 0,Y 395.777,Z 476.134,A -85,B 0,C 180,E1 -11245.927,E2 -11245.927} C_VEL
LIN {X 0,Y 395.763,Z 478.579,A -85,B 0,C 180,E1 -11247.965,E2 -11247.965} C_VEL
LIN {X 0,Y 395.792,Z 479.168,A -85,B 0,C 180,E1 -11248.983,E2 -11248.983} C_VEL
LIN {X 0,Y 395.792,Z 479.168,A -85,B 0,C 180,E1 -11251.017,E2 -11251.017} C_VEL
LIN {X 0,Y 395.763,Z 478.579,A -85,B 0,C 180,E1 -11252.035,E2 -11252.035} C_VEL
LIN {X 0,Y 395.777,Z 476.134,A -85,B 0,C 180,E1 -11254.073,E2 -11254.073} C_VEL
LIN {X 0,Y 395.848,Z 474.337,A -85,B 0,C 180,E1 -11255.093,E2 -11255.093} C_VEL
LIN {X 0,Y 395.922,Z 470.73,A -85,B 0,C 180,E1 -11256.625,E2 -11256.625} C_VEL
LIN {X 0,Y 396.228,Z 465.985,A -85,B 0,C 180,E1 -11258.158,E2 -11258.158} C_VEL
LIN {X 0,Y 396.62,Z 459.962,A -85,B 0,C 180,E1 -11259.691,E2 -11259.691} C_VEL
LIN {X 0,Y 397.067,Z 453.864,A -85,B 0,C 180,E1 -11260.969,E2 -11260.969} C_VEL
LIN {X 0,Y 397.6,Z 448.165,A -85,B 0,C 180,E1 -11261.987,E2 -11261.987} C_VEL
LIN {X 0,Y 398.301,Z 439.609,A -85,B 0,C 180,E1 -11263.261,E2 -11263.261} C_VEL
LIN {X 0,Y 398.935,Z 431.426,A -85,B 0,C 180,E1 -11264.278,E2 -11264.278} C_VEL
LIN {X 0,Y 399.588,Z 423.048,A -85,B 0,C 180,E1 -11265.153,E2 -11265.153} C_VEL
LIN {X 0,Y 400.306,Z 414.196,A -85,B 0,C 180,E1 -11265.922,E2 -11265.922} C_VEL
LIN {X 0,Y 400.893,Z 404.866,A -85,B 0,C 180,E1 -11266.589,E2 -11266.589} C_VEL
LIN {X 0,Y 399.679,Z 394.599,A -85,B 0,C 180,E1 -11267.246,E2 -11267.246} C_VEL
LIN {X 0,Y 398.041,Z 384.737,A -85,B 0,C 180,E1 -11267.765,E2 -11267.765} C_VEL
LIN {X 0,Y 395.925,Z 374.094,A -85,B 0,C 180,E1 -11268.228,E2 -11268.228} C_VEL
LIN {X 0,Y 396.067,Z 370.203,A -85,B 0,C 180,E1 -11270.787,E2 -11270.787} C_VEL
LIN {X 0,Y 396.298,Z 365.282,A -85,B 0,C 180,E1 -11274.072,E2 -11274.072} C_VEL
LIN {X 0,Y 396.674,Z 360.086,A -85,B 0,C 180,E1 -11277.641,E2 -11277.641} C_VEL
LIN {X 0,Y 397.009,Z 355.55,A -85,B 0,C 180,E1 -11280.888,E2 -11280.888} C_VEL
LIN {X 0,Y 397.385,Z 350.786,A -85,B 0,C 180,E1 -11284.467,E2 -11284.467} C_VEL
LIN {X 0,Y 397.816,Z 346.073,A -85,B 0,C 180,E1 -11288.194,E2 -11288.194} C_VEL
LIN {X 0,Y 398.058,Z 343.021,A -85,B 0,C 180,E1 -11290.788,E2 -11290.788} C_VEL
LIN {X 0,Y 398.074,Z 339.886,A -85,B 0,C 180,E1 -11293.626,E2 -11293.626} C_VEL
LIN {X 0,Y 397.753,Z 337.027,A -85,B 0,C 180,E1 -11296.44,E2 -11296.44} C_VEL
LIN {X 0,Y 397.359,Z 334.16,A -85,B 0,C 180,E1 -11299.511,E2 -11299.511} C_VEL
LIN {X 0,Y 397.14,Z 332.741,A -85,B 0,C 180,E1 -11301.137,E2 -11301.137} C_VEL
LIN {X 0,Y 397.12,Z 332.523,A -85,B 0,C 180,E1 -11304.496,E2 -11304.496} C_VEL
LIN {X 0,Y 397.08,Z 332.526,A -85,B 0,C 180,E1 -11307.928,E2 -11307.928} C_VEL
LIN {X 0,Y 397.123,Z 332.516,A -85,B 0,C 180,E1 -11311.456,E2 -11311.456} C_VEL
LIN {X 0,Y 397.153,Z 332.511,A -85,B 0,C 180,E1 -11314.487,E2 -11314.487} C_VEL
LIN {X 0,Y 397.096,Z 332.519,A -85,B 0,C 180,E1 -11318.181,E2 -11318.181} C_VEL
LIN {X 0,Y 397.158,Z 332.514,A -85,B 0,C 180,E1 -11321.426,E2 -11321.426} C_VEL
LIN {X 0,Y 397.179,Z 332.507,A -85,B 0,C 180,E1 -11324.607,E2 -11324.607} C_VEL
LIN {X 0,Y 397.219,Z 332.506,A -85,B 0,C 180,E1 -11327.741,E2 -11327.741} C_VEL
LIN {X 0,Y 397.253,Z 332.499,A -85,B 0,C 180,E1 -11330.838,E2 -11330.838} C_VEL
LIN {X 0,Y 397.37,Z 332.484,A -85,B 0,C 180,E1 -11333.908,E2 -11333.908} C_VEL
LIN {X 0,Y 397.45,Z 332.473,A -85,B 0,C 180,E1 -11337.973,E2 -11337.973} C_VEL
LIN {X 0,Y 397.578,Z 332.457,A -85,B 0,C 180,E1 -11339.999,E2 -11339.999} C_VEL
LIN {X 0,Y 397.38,Z 332.488,A -85,B 0,C 180,E1 -11343.041,E2 -11343.041} C_VEL
LIN {X 0,Y 397.344,Z 332.487,A -85,B 0,C 180,E1 -11346.557,E2 -11346.557} C_VEL
LIN {X 0,Y 397.252,Z 332.502,A -85,B 0,C 180,E1 -11349.161,E2 -11349.161} C_VEL
LIN {X 0,Y 397.218,Z 332.503,A -85,B 0,C 180,E1 -11352.258,E2 -11352.258} C_VEL
LIN {X 0,Y 397.177,Z 332.508,A -85,B 0,C 180,E1 -11355.391,E2 -11355.391} C_VEL
LIN {X 0,Y 397.16,Z 332.514,A -85,B 0,C 180,E1 -11358.573,E2 -11358.573} C_VEL
LIN {X 0,Y 397.093,Z 332.518,A -85,B 0,C 180,E1 -11361.818,E2 -11361.818} C_VEL
LIN {X 0,Y 397.15,Z 332.51,A -85,B 0,C 180,E1 -11365.512,E2 -11365.512} C_VEL
LIN {X 0,Y 397.12,Z 332.521,A -85,B 0,C 180,E1 -11368.543,E2 -11368.543} C_VEL
LIN {X 0,Y 397.075,Z 332.523,A -85,B 0,C 180,E1 -11372.071,E2 -11372.071} C_VEL
LIN {X 0,Y 397.117,Z 332.515,A -85,B 0,C 180,E1 -11375.503,E2 -11375.503} C_VEL
LIN {X 0,Y 397.133,Z 332.513,A -85,B 0,C 180,E1 -11378.862,E2 -11378.862} C_VEL
LIN {X 0,Y 397.156,Z 332.516,A -85,B 0,C 180,E1 -11382.255,E2 -11382.255} C_VEL
LIN {X 0,Y 397.109,Z 332.516,A -85,B 0,C 180,E1 -11385.065,E2 -11385.065} C_VEL
LIN {X 0,Y 397.106,Z 332.523,A -85,B 0,C 180,E1 -11388.014,E2 -11388.014} C_VEL
LIN {X 0,Y 397.133,Z 332.513,A -85,B 0,C 180,E1 -11391.137,E2 -11391.137} C_VEL
LIN {X 0,Y 397.116,Z 332.516,A -85,B 0,C 180,E1 -11394.496,E2 -11394.496} C_VEL
LIN {X 0,Y 397.075,Z 332.525,A -85,B 0,C 180,E1 -11397.928,E2 -11397.928} C_VEL
LIN {X 0,Y 397.119,Z 332.519,A -85,B 0,C 180,E1 -11401.456,E2 -11401.456} C_VEL
LIN {X 0,Y 397.149,Z 332.511,A -85,B 0,C 180,E1 -11404.487,E2 -11404.487} C_VEL
LIN {X 0,Y 397.105,Z 332.518,A -85,B 0,C 180,E1 -11407.086,E2 -11407.086} C_VEL
LIN {X 0,Y 397.145,Z 332.513,A -85,B 0,C 180,E1 -11410.353,E2 -11410.353} C_VEL
LIN {X 0,Y 397.163,Z 332.515,A -85,B 0,C 180,E1 -11413.553,E2 -11413.553} C_VEL
LIN {X 0,Y 397.225,Z 332.507,A -85,B 0,C 180,E1 -11416.703,E2 -11416.703} C_VEL
LIN {X 0,Y 397.215,Z 332.508,A -85,B 0,C 180,E1 -11419.809,E2 -11419.809} C_VEL
LIN {X 0,Y 397.361,Z 332.489,A -85,B 0,C 180,E1 -11422.888,E2 -11422.888} C_VEL
LIN {X 0,Y 397.253,Z 332.504,A -85,B 0,C 180,E1 -11424.925,E2 -11424.925} C_VEL
LIN {X 0,Y 397.448,Z 332.477,A -85,B 0,C 180,E1 -11427.973,E2 -11427.973} C_VEL
LIN {X 0,Y 397.578,Z 332.463,A -85,B 0,C 180,E1 -11430,E2 -11430} C_VEL
LIN {X 0,Y 397.378,Z 332.487,A -85,B 0,C 180,E1 -11433.041,E2 -11433.041} C_VEL
LIN {X 0,Y 397.361,Z 332.489,A -85,B 0,C 180,E1 -11437.112,E2 -11437.112} C_VEL
LIN {X 0,Y 397.215,Z 332.508,A -85,B 0,C 180,E1 -11440.191,E2 -11440.191} C_VEL
LIN {X 0,Y 397.223,Z 332.507,A -85,B 0,C 180,E1 -11443.321,E2 -11443.321} C_VEL
LIN {X 0,Y 397.178,Z 332.513,A -85,B 0,C 180,E1 -11447.155,E2 -11447.155} C_VEL
LIN {X 0,Y 397.11,Z 332.52,A -85,B 0,C 180,E1 -11450.729,E2 -11450.729} C_VEL
LIN {X 0,Y 397.129,Z 332.516,A -85,B 0,C 180,E1 -11454.018,E2 -11454.018} C_VEL
LIN {X 0,Y 397.131,Z 332.518,A -85,B 0,C 180,E1 -11456.31,E2 -11456.31} C_VEL
LIN {X 0,Y 396.46,Z 332.597,A -85,B 0,C 180,E1 -11457.156,E2 -11457.156} C_VEL
LIN {X 0,Y 393.586,Z 332.959,A -85,B 0,C 180,E1 -11458.532,E2 -11458.532} C_VEL
LIN {X 0,Y 391.149,Z 333.264,A -85,B 0,C 180,E1 -11459.643,E2 -11459.643} C_VEL
LIN {X 0,Y 390.096,Z 333.393,A -85,B 0,C 180,E1 -11460.503,E2 -11460.503} C_VEL
LIN {X 0,Y 390.008,Z 333.402,A -85,B 0,C 180,E1 -11460.794,E2 -11460.794} C_VEL
LIN {X 0,Y 390.064,Z 333.398,A -85,B 0,C 180,E1 -11464.025,E2 -11464.025} C_VEL
LIN {X 0,Y 390.043,Z 333.397,A -85,B 0,C 180,E1 -11467.552,E2 -11467.552} C_VEL
LIN {X 0,Y 390.073,Z 333.392,A -85,B 0,C 180,E1 -11470.825,E2 -11470.825} C_VEL
LIN {X 0,Y 390.057,Z 333.4,A -85,B 0,C 180,E1 -11473.887,E2 -11473.887} C_VEL
LIN {X 0,Y 390.112,Z 333.387,A -85,B 0,C 180,E1 -11476.798,E2 -11476.798} C_VEL
LIN {X 0,Y 390.074,Z 333.396,A -85,B 0,C 180,E1 -11479.564,E2 -11479.564} C_VEL
LIN {X 0,Y 390.043,Z 333.396,A -85,B 0,C 180,E1 -11482.449,E2 -11482.449} C_VEL
LIN {X 0,Y 390.065,Z 333.396,A -85,B 0,C 180,E1 -11486.046,E2 -11486.046} C_VEL
LIN {X 0,Y 390.043,Z 333.399,A -85,B 0,C 180,E1 -11489.869,E2 -11489.869} C_VEL
LIN {X 0,Y 390.111,Z 333.391,A -85,B 0,C 180,E1 -11493.232,E2 -11493.232} C_VEL
LIN {X 0,Y 390.074,Z 333.393,A -85,B 0,C 180,E1 -11496.761,E2 -11496.761} C_VEL
LIN {X 0,Y 390.102,Z 333.389,A -85,B 0,C 180,E1 -11499.984,E2 -11499.984} C_VEL
LIN {X 0,Y 390.136,Z 333.391,A -85,B 0,C 180,E1 -11503.249,E2 -11503.249} C_VEL
LIN {X 0,Y 390.193,Z 333.378,A -85,B 0,C 180,E1 -11506.562,E2 -11506.562} C_VEL
LIN {X 0,Y 390.204,Z 333.379,A -85,B 0,C 180,E1 -11510.672,E2 -11510.672} C_VEL
LIN {X 0,Y 390.323,Z 333.361,A -85,B 0,C 180,E1 -11513.799,E2 -11513.799} C_VEL
LIN {X 0,Y 390.42,Z 333.349,A -85,B 0,C 180,E1 -11517.937,E2 -11517.937} C_VEL
LIN {X 0,Y 390.547,Z 333.333,A -85,B 0,C 180,E1 -11520.001,E2 -11520.001} C_VEL
LIN {X 0,Y 390.313,Z 333.365,A -85,B 0,C 180,E1 -11523.097,E2 -11523.097} C_VEL
LIN {X 0,Y 390.324,Z 333.363,A -85,B 0,C 180,E1 -11526.203,E2 -11526.203} C_VEL
LIN {X 0,Y 390.205,Z 333.376,A -85,B 0,C 180,E1 -11529.329,E2 -11529.329} C_VEL
LIN {X 0,Y 390.194,Z 333.377,A -85,B 0,C 180,E1 -11533.439,E2 -11533.439} C_VEL
LIN {X 0,Y 390.129,Z 333.385,A -85,B 0,C 180,E1 -11537.299,E2 -11537.299} C_VEL
LIN {X 0,Y 390.093,Z 333.395,A -85,B 0,C 180,E1 -11540.473,E2 -11540.473} C_VEL
LIN {X 0,Y 390.078,Z 333.395,A -85,B 0,C 180,E1 -11544.481,E2 -11544.481} C_VEL
LIN {X 0,Y 390.118,Z 333.391,A -85,B 0,C 180,E1 -11547.931,E2 -11547.931} C_VEL
LIN {X 0,Y 390.024,Z 333.4,A -85,B 0,C 180,E1 -11551.505,E2 -11551.505} C_VEL
LIN {X 0,Y 390.086,Z 333.392,A -85,B 0,C 180,E1 -11555.207,E2 -11555.207} C_VEL
LIN {X 0,Y 390.045,Z 333.402,A -85,B 0,C 180,E1 -11557.78,E2 -11557.78} C_VEL
LIN {X 0,Y 390.193,Z 334.213,A -85,B 0,C 180,E1 -11559.241,E2 -11559.241} C_VEL
LIN {X 0,Y 390.592,Z 337.083,A -85,B 0,C 180,E1 -11562.463,E2 -11562.463} C_VEL
LIN {X 0,Y 391.01,Z 340.516,A -85,B 0,C 180,E1 -11565.969,E2 -11565.969} C_VEL
LIN {X 0,Y 391.05,Z 343.026,A -85,B 0,C 180,E1 -11568.32,E2 -11568.32} C_VEL
LIN {X 0,Y 390.869,Z 346.086,A -85,B 0,C 180,E1 -11571.001,E2 -11571.001} C_VEL
LIN {X 0,Y 390.512,Z 349.815,A -85,B 0,C 180,E1 -11574.083,E2 -11574.083} C_VEL
LIN {X 0,Y 390.148,Z 353.888,A -85,B 0,C 180,E1 -11577.289,E2 -11577.289} C_VEL
LIN {X 0,Y 389.72,Z 358.685,A -85,B 0,C 180,E1 -11580.863,E2 -11580.863} C_VEL
LIN {X 0,Y 389.377,Z 363.531,A -85,B 0,C 180,E1 -11584.33,E2 -11584.33} C_VEL
LIN {X 0,Y 389.112,Z 368.425,A -85,B 0,C 180,E1 -11587.71,E2 -11587.71} C_VEL
LIN {X 0,Y 388.855,Z 373.344,A -85,B 0,C 180,E1 -11591.015,E2 -11591.015} C_VEL
LIN {X 0,Y 388.847,Z 374.147,A -85,B 0,C 180,E1 -11591.459,E2 -11591.459} C_VEL
LIN {X 0,Y 391.045,Z 384.841,A -85,B 0,C 180,E1 -11591.918,E2 -11591.918} C_VEL
LIN {X 0,Y 392.824,Z 395.418,A -85,B 0,C 180,E1 -11592.496,E2 -11592.496} C_VEL
LIN {X 0,Y 393.801,Z 403.454,A -85,B 0,C 180,E1 -11593.024,E2 -11593.024} C_VEL
LIN {X 0,Y 393.849,Z 409.102,A -85,B 0,C 180,E1 -11593.411,E2 -11593.411} C_VEL
LIN {X 0,Y 393.007,Z 420.014,A -85,B 0,C 180,E1 -11594.308,E2 -11594.308} C_VEL
LIN {X 0,Y 392.205,Z 428.959,A -85,B 0,C 180,E1 -11595.206,E2 -11595.206} C_VEL
LIN {X 0,Y 391.617,Z 436.302,A -85,B 0,C 180,E1 -11596.08,E2 -11596.08} C_VEL
LIN {X 0,Y 390.936,Z 444.714,A -85,B 0,C 180,E1 -11597.278,E2 -11597.278} C_VEL
LIN {X 0,Y 390.317,Z 450.915,A -85,B 0,C 180,E1 -11598.313,E2 -11598.313} C_VEL
LIN {X 0,Y 389.798,Z 457.455,A -85,B 0,C 180,E1 -11599.613,E2 -11599.613} C_VEL
LIN {X 0,Y 389.433,Z 461.957,A -85,B 0,C 180,E1 -11600.653,E2 -11600.653} C_VEL
LIN {X 0,Y 389.044,Z 467.449,A -85,B 0,C 180,E1 -11602.213,E2 -11602.213} C_VEL
LIN {X 0,Y 388.798,Z 471.895,A -85,B 0,C 180,E1 -11603.826,E2 -11603.826} C_VEL
LIN {X 0,Y 388.745,Z 474.14,A -85,B 0,C 180,E1 -11604.814,E2 -11604.814} C_VEL
LIN {X 0,Y 388.702,Z 475.939,A -85,B 0,C 180,E1 -11605.853,E2 -11605.853} C_VEL
LIN {X 0,Y 388.662,Z 478.383,A -85,B 0,C 180,E1 -11607.927,E2 -11607.927} C_VEL
LIN {X 0,Y 388.704,Z 478.972,A -85,B 0,C 180,E1 -11608.964,E2 -11608.964} C_VEL
LIN {X 0,Y 388.704,Z 478.972,A -85,B 0,C 180,E1 -11611.036,E2 -11611.036} C_VEL
LIN {X 0,Y 388.662,Z 478.383,A -85,B 0,C 180,E1 -11612.073,E2 -11612.073} C_VEL
LIN {X 0,Y 388.702,Z 475.939,A -85,B 0,C 180,E1 -11614.147,E2 -11614.147} C_VEL
LIN {X 0,Y 388.729,Z 472.876,A -85,B 0,C 180,E1 -11615.755,E2 -11615.755} C_VEL
LIN {X 0,Y 388.942,Z 469.002,A -85,B 0,C 180,E1 -11617.267,E2 -11617.267} C_VEL
LIN {X 0,Y 389.293,Z 463.873,A -85,B 0,C 180,E1 -11618.827,E2 -11618.827} C_VEL
LIN {X 0,Y 389.67,Z 458.61,A -85,B 0,C 180,E1 -11620.128,E2 -11620.128} C_VEL
LIN {X 0,Y 390.177,Z 452.291,A -85,B 0,C 180,E1 -11621.428,E2 -11621.428} C_VEL
LIN {X 0,Y 390.772,Z 446.341,A -85,B 0,C 180,E1 -11622.464,E2 -11622.464} C_VEL
LIN {X 0,Y 391.341,Z 439.411,A -85,B 0,C 180,E1 -11623.501,E2 -11623.501} C_VEL
LIN {X 0,Y 392.017,Z 431.229,A -85,B 0,C 180,E1 -11624.536,E2 -11624.536} C_VEL
LIN {X 0,Y 392.722,Z 422.716,A -85,B 0,C 180,E1 -11625.438,E2 -11625.438} C_VEL
LIN {X 0,Y 393.483,Z 414,A -85,B 0,C 180,E1 -11626.205,E2 -11626.205} C_VEL
LIN {X 0,Y 394.003,Z 404.916,A -85,B 0,C 180,E1 -11626.871,E2 -11626.871} C_VEL
LIN {X 0,Y 392.867,Z 395.842,A -85,B 0,C 180,E1 -11627.48,E2 -11627.48} C_VEL
LIN {X 0,Y 391.128,Z 385.234,A -85,B 0,C 180,E1 -11628.063,E2 -11628.063} C_VEL
LIN {X 0,Y 388.871,Z 373.924,A -85,B 0,C 180,E1 -11628.571,E2 -11628.571} C_VEL
LIN {X 0,Y 389.012,Z 370.063,A -85,B 0,C 180,E1 -11631.182,E2 -11631.182} C_VEL
LIN {X 0,Y 389.256,Z 365.14,A -85,B 0,C 180,E1 -11634.536,E2 -11634.536} C_VEL
LIN {X 0,Y 389.634,Z 360.284,A -85,B 0,C 180,E1 -11637.968,E2 -11637.968} C_VEL
LIN {X 0,Y 390.017,Z 355.472,A -85,B 0,C 180,E1 -11641.505,E2 -11641.505} C_VEL
LIN {X 0,Y 390.302,Z 352.121,A -85,B 0,C 180,E1 -11644.075,E2 -11644.075} C_VEL
LIN {X 0,Y 390.728,Z 347.607,A -85,B 0,C 180,E1 -11647.702,E2 -11647.702} C_VEL
LIN {X 0,Y 391.026,Z 343.791,A -85,B 0,C 180,E1 -11650.985,E2 -11650.985} C_VEL
LIN {X 0,Y 391.064,Z 341.502,A -85,B 0,C 180,E1 -11653.072,E2 -11653.072} C_VEL
LIN {X 0,Y 390.773,Z 338.544,A -85,B 0,C 180,E1 -11656.004,E2 -11656.004} C_VEL
LIN {X 0,Y 390.355,Z 335.218,A -85,B 0,C 180,E1 -11659.597,E2 -11659.597} C_VEL
LIN {X 0,Y 390.157,Z 334.081,A -85,B 0,C 180,E1 -11660.915,E2 -11660.915} C_VEL
LIN {X 0,Y 390.045,Z 333.402,A -85,B 0,C 180,E1 -11662.449,E2 -11662.449} C_VEL
LIN {X 0,Y 390.069,Z 333.399,A -85,B 0,C 180,E1 -11666.045,E2 -11666.045} C_VEL
LIN {X 0,Y 390.047,Z 333.402,A -85,B 0,C 180,E1 -11669.868,E2 -11669.868} C_VEL
LIN {X 0,Y 390.114,Z 333.388,A -85,B 0,C 180,E1 -11673.231,E2 -11673.231} C_VEL
LIN {X 0,Y 390.068,Z 333.393,A -85,B 0,C 180,E1 -11676.763,E2 -11676.763} C_VEL
LIN {X 0,Y 390.106,Z 333.391,A -85,B 0,C 180,E1 -11679.983,E2 -11679.983} C_VEL
LIN {X 0,Y 390.138,Z 333.387,A -85,B 0,C 180,E1 -11683.248,E2 -11683.248} C_VEL
LIN {X 0,Y 390.194,Z 333.377,A -85,B 0,C 180,E1 -11686.561,E2 -11686.561} C_VEL
LIN {X 0,Y 390.205,Z 333.376,A -85,B 0,C 180,E1 -11690.671,E2 -11690.671} C_VEL
LIN {X 0,Y 390.324,Z 333.363,A -85,B 0,C 180,E1 -11693.797,E2 -11693.797} C_VEL
LIN {X 0,Y 390.419,Z 333.35,A -85,B 0,C 180,E1 -11697.936,E2 -11697.936} C_VEL
LIN {X 0,Y 390.547,Z 333.333,A -85,B 0,C 180,E1 -11699.999,E2 -11699.999} C_VEL
LIN {X 0,Y 390.314,Z 333.369,A -85,B 0,C 180,E1 -11703.096,E2 -11703.096} C_VEL
LIN {X 0,Y 390.301,Z 333.363,A -85,B 0,C 180,E1 -11706.551,E2 -11706.551} C_VEL
LIN {X 0,Y 390.204,Z 333.379,A -85,B 0,C 180,E1 -11709.328,E2 -11709.328} C_VEL
LIN {X 0,Y 390.193,Z 333.378,A -85,B 0,C 180,E1 -11713.438,E2 -11713.438} C_VEL
LIN {X 0,Y 390.147,Z 333.384,A -85,B 0,C 180,E1 -11717.307,E2 -11717.307} C_VEL
LIN {X 0,Y 390.085,Z 333.395,A -85,B 0,C 180,E1 -11720.47,E2 -11720.47} C_VEL
LIN {X 0,Y 390.076,Z 333.397,A -85,B 0,C 180,E1 -11724.48,E2 -11724.48} C_VEL
LIN {X 0,Y 390.114,Z 333.388,A -85,B 0,C 180,E1 -11727.93,E2 -11727.93} C_VEL
LIN {X 0,Y 390.02,Z 333.399,A -85,B 0,C 180,E1 -11731.504,E2 -11731.504} C_VEL
LIN {X 0,Y 390.065,Z 333.396,A -85,B 0,C 180,E1 -11734.024,E2 -11734.024} C_VEL
LIN {X 0,Y 390.044,Z 333.396,A -85,B 0,C 180,E1 -11737.551,E2 -11737.551} C_VEL
LIN {X 0,Y 390.079,Z 333.392,A -85,B 0,C 180,E1 -11740.826,E2 -11740.826} C_VEL
LIN {X 0,Y 390.1,Z 333.393,A -85,B 0,C 180,E1 -11743.893,E2 -11743.893} C_VEL
LIN {X 0,Y 390.077,Z 333.394,A -85,B 0,C 180,E1 -11747.619,E2 -11747.619} C_VEL
LIN {X 0,Y 390.091,Z 333.39,A -85,B 0,C 180,E1 -11750.908,E2 -11750.908} C_VEL
LIN {X 0,Y 390.082,Z 333.391,A -85,B 0,C 180,E1 -11754.793,E2 -11754.793} C_VEL
LIN {X 0,Y 390.028,Z 333.403,A -85,B 0,C 180,E1 -11757.875,E2 -11757.875} C_VEL
LIN {X 0,Y 390.055,Z 333.395,A -85,B 0,C 180,E1 -11760.89,E2 -11760.89} C_VEL
LIN {X 0,Y 390.115,Z 333.388,A -85,B 0,C 180,E1 -11764.256,E2 -11764.256} C_VEL
LIN {X 0,Y 390.037,Z 333.401,A -85,B 0,C 180,E1 -11767.766,E2 -11767.766} C_VEL
LIN {X 0,Y 390.102,Z 333.394,A -85,B 0,C 180,E1 -11771.078,E2 -11771.078} C_VEL
LIN {X 0,Y 390.136,Z 333.389,A -85,B 0,C 180,E1 -11774.323,E2 -11774.323} C_VEL
LIN {X 0,Y 390.167,Z 333.385,A -85,B 0,C 180,E1 -11777.517,E2 -11777.517} C_VEL
LIN {X 0,Y 390.311,Z 333.367,A -85,B 0,C 180,E1 -11781.718,E2 -11781.718} C_VEL
LIN {X 0,Y 390.35,Z 333.563,A -85,B 0,C 180,E1 -11782.704,E2 -11782.704} C_VEL
LIN {X 0,Y 390.912,Z 335.476,A -85,B 0,C 180,E1 -11783.159,E2 -11783.159} C_VEL
LIN {X 0,Y 392.539,Z 337.757,A -85,B 0,C 180,E1 -11784.349,E2 -11784.349} C_VEL
LIN {X 0,Y 394.308,Z 339.018,A -85,B 0,C 180,E1 -11785.912,E2 -11785.912} C_VEL
LIN {X 0,Y 395.197,Z 339.225,A -85,B 0,C 180,E1 -11786.942,E2 -11786.942} C_VEL
LIN {X 0,Y 396.207,Z 339.464,A -85,B 0,C 180,E1 -11788.984,E2 -11788.984} C_VEL
LIN {X 0,Y 396.373,Z 339.46,A -85,B 0,C 180,E1 -11790,E2 -11790} C_VEL
LIN {X 0,Y 395.808,Z 339.385,A -85,B 0,C 180,E1 -11792.035,E2 -11792.035} C_VEL
LIN {X 0,Y 394.474,Z 339.066,A -85,B 0,C 180,E1 -11793.894,E2 -11793.894} C_VEL
LIN {X 0,Y 392.691,Z 337.905,A -85,B 0,C 180,E1 -11795.52,E2 -11795.52} C_VEL
LIN {X 0,Y 390.995,Z 335.651,A -85,B 0,C 180,E1 -11796.774,E2 -11796.774} C_VEL
LIN {X 0,Y 390.385,Z 333.728,A -85,B 0,C 180,E1 -11797.268,E2 -11797.268} C_VEL
LIN {X 0,Y 390.316,Z 333.368,A -85,B 0,C 180,E1 -11797.353,E2 -11797.353} C_VEL
LIN {X 0,Y 390.165,Z 333.385,A -85,B 0,C 180,E1 -11800.377,E2 -11800.377} C_VEL
LIN {X 0,Y 390.166,Z 333.385,A -85,B 0,C 180,E1 -11803.542,E2 -11803.542} C_VEL
LIN {X 0,Y 390.145,Z 333.388,A -85,B 0,C 180,E1 -11807.308,E2 -11807.308} C_VEL
LIN {X 0,Y 390.089,Z 333.397,A -85,B 0,C 180,E1 -11810.472,E2 -11810.472} C_VEL
LIN {X 0,Y 390.086,Z 333.391,A -85,B 0,C 180,E1 -11813.351,E2 -11813.351} C_VEL
LIN {X 0,Y 390.11,Z 333.39,A -85,B 0,C 180,E1 -11816.768,E2 -11816.768} C_VEL
LIN {X 0,Y 390.035,Z 333.403,A -85,B 0,C 180,E1 -11820.3,E2 -11820.3} C_VEL
LIN {X 0,Y 390.008,Z 333.402,A -85,B 0,C 180,E1 -11820.794,E2 -11820.794} C_VEL
LIN {X 0,Y 389.334,Z 333.487,A -85,B 0,C 180,E1 -11821.657,E2 -11821.657} C_VEL
LIN {X 0,Y 386.487,Z 333.839,A -85,B 0,C 180,E1 -11823.058,E2 -11823.058} C_VEL
LIN {X 0,Y 384.09,Z 334.144,A -85,B 0,C 180,E1 -11824.191,E2 -11824.191} C_VEL
LIN {X 0,Y 383.072,Z 334.265,A -85,B 0,C 180,E1 -11825.067,E2 -11825.067} C_VEL
LIN {X 0,Y 382.995,Z 334.274,A -85,B 0,C 180,E1 -11825.364,E2 -11825.364} C_VEL
LIN {X 0,Y 383.005,Z 334.274,A -85,B 0,C 180,E1 -11828.6,E2 -11828.6} C_VEL
LIN {X 0,Y 383.01,Z 334.273,A -85,B 0,C 180,E1 -11831.344,E2 -11831.344} C_VEL
